SYMBOL_TABLE
"$Revision: 1.101 $"		BOOL	//      $Date: 2008/12/01 14:04:16CET $ $Author: hgc $
"Z_Umlaufzaehler"	C 1	COUNTER	// Temp_Fb242
"Z_Impulszaehler_Motor"	C 9	COUNTER
"Z_min_Takt_Vlies"	C 20	COUNTER	// Minutenzähler für Zwangstakt Vlies
"Z_sec_Takt_Vlies"	C 21	COUNTER	// Sekundenzähler für Zwangstakt Vlies
"Z_MIN_TAKT_SPALTSIEB"	C 22	COUNTER	// Minutenzähler für Intervallbetrieb Spaltsieb
"Z_SEC_TAKT_SPALTSIEB"	C 23	COUNTER	// Sekundenzähler für Intervallbetrieb Spaltsieb
"Z_SPALTSIEB_TAKTE"	C 24	COUNTER	// Zähler für die Spaltsiebtakte
"Z_MSST_COUNT"	C 30	COUNTER
"Z_Schm_FD_War"	C 57	COUNTER
"DB_PLC_MESSAGE"	DB 2	UDT 2	// Schnittstelle für Alarme und Meldungen
"DB_SIEM_GP_DB3"	DB 3	DB 3	// GP SIEMENS
"DB_ALARM_KENNUNG"	DB 4	DB 4	// Siemens Grundprogramm
"DB_SIEM_GP_DB5"	DB 5	DB 5	// GP SIEMENS
"DB_SIEM_GP_DB6"	DB 6	DB 6	// GP SIEMENS
"DB_SIEM_STARTUP"	DB 7	FB 1	// Baseprogram Start-up
"DB_SIEM_SYSTEM4"	DB 8	DB 8	// Baseprogram System
"DB_SIEM_NCK"	DB 10	UDT 10	// Interface NCK
"DB_SIEM_BAG"	DB 11	UDT 11	// Interface BAG
"DB_SINRPC"	DB 12	DB 12	// Interface RPC-PLC
"DB_SIEM_INSTANZ_DB_FB6"	DB 15	FB 6	// GP SIEMENS: Instanz-DB zu FB6
"DB_SIEM_PI"	DB 16	DB 16	// Interface PI-Services
"DB_SIEM_VERSION_CODE"	DB 17	DB 17	// GP SIEMENS: Versionskennung
"DB_SPL"	DB 18	DB 18	// SPL Daten
"DB_SIEM_MMC"	DB 19	UDT 19	// Schnittstelle MMC-Signale
"DB_PLC_MD_DB20"	DB 20	UDT 20	// Maschinenparameter
"DB_SIEM_KANAL_1"	DB 21	UDT 21	// Interface Chanel 1
"DB_SIEM_KANAL_2"	DB 22	UDT 21	// Interface Chanel 2
"DB_ACHSE1_X"	DB 31	UDT 31	// Interface Axis 1 X
"DB_ACHSE2_Y"	DB 32	UDT 31	// Interface Axis 2 Y
"DB_ACHSE3_Z"	DB 33	UDT 31	// Interface Axis 3 Z
"DB_ACHSE4"	DB 34	UDT 31	// Interface Axis 4
"DB_ACHSE5"	DB 35	UDT 31	// Interface Axis 5
"DB_ACHSE6_SPINDEL"	DB 36	UDT 31	// Interface Axis 6 Spindel
"DB_ACHSE7"	DB 37	UDT 31	// Interface Axis 7
"DB_ACHSE8"	DB 38	UDT 31	// Interface Axis 8
"DB_ACHSE9"	DB 39	UDT 31	// Interface Axis 9
"DB_ACHSE10"	DB 40	UDT 31	// Interface Axis 10
"DB_ACHSE11"	DB 41	UDT 31	// Interface Axis 11
"DB_ACHSE12"	DB 42	UDT 31	// Interface Axis 12
"DB_ACHSE13"	DB 43	UDT 31	// Interface Axis 13
"DB_ACHSE14"	DB 44	UDT 31	// Interface Axis 14
"DB_ACHSE15"	DB 45	UDT 31	// Interface Axis 15
"DB_ACHSE16"	DB 46	UDT 31	// Interface Axis 16
"DB_ACHSE17"	DB 47	UDT 31	// Achs Nahtstelle (Achse 17) Simulierte Z-Achse für Komet (U-Achse)
"DB_ACHSE18"	DB 48	UDT 31	// Interface Axis 18
"DB_ACHSE19"	DB 49	UDT 31	// Interface Axis 19
"DB_HR"	DB 50	DB 50	// HR Datenbaustein
"DB_HMI_OEM"	DB 57	DB 57	// OEM Datenbaustein
"DB_HMI"	DB 59	UDT 59	// HMI PRO Datenbaustein
"DB_DEC_HMI"	DB 62	DB 62	// DEC HMI Datenbaustein
"DB_FAMILIEN_MODUL"	DB 65	UDT 65	// Datenbaustein Familienmodul
"DB_TIMER"	DB 66	DB 66	// DB für Timerbaustein
"DB_NC_PLC"	DB 70	UDT 70	// DB für DUAL-Port-RAM: Datentausch NC<==>PLC
"TMLoadIF"	DB 71	UDT 71	// Interface loading-/unloadingstation for Toolmanagment
"TMSpindleIF"	DB 72	UDT 72	// Schnittstelle: Werkzeugverw.: Wechsel in Spindel
"Revolver"	DB 73	UDT 73	// Interface Revolver for Toolmanagment
"DB_OVR_WANDLER"	DB 75	DB 75	// Overridewandler
"DB_DP_DIAG_SINUMERIK"	DB 78	DB 78	// DB DP-Diagnose Sinumerik mit Wizard
"DI_FB_DETAIL_DP_DIAG"	DB 79	FB 96	// Instanz-DB zu FB96
"DB_CMM_PLC"	DB 82	DB 82	// SM PLC-Interface
"DI_FB_PLC_Absturz_GP"	DB 90	FB 29	// Instanz-DB für Diagnose PLC-Absturz im Grundprogramm
"DB_PLC_ABSTURZ_GP_RING"	DB 91	DB 91	// PLC Absturz Grundprogramm
"DB_SIEM_DB_DIAG_DETAIL"	DB 96	FB 96	// Instanz-DB zu FB96 (Transline 200 Anzeige)
"DB_HMI_PRO_RANG_DIAG"	DB 97	DB 97	// Rangierung Diagnosedaten integrierte CP auf HMI-PRO
"DB_DM_PLC_VERSION"	DB 99	DB 99	// Plc Version
"DB_REMANENT"	DB 100	UDT 100	// Remanente Daten
"DB_OEM"	DB 101	DB 101	// OEM-Daten 1
"DB_FEHLERMELDUNG"	DB 102	DB 102	// Fehler- Betriebsmeldungen Maschine
"DB_ANWENDER_SOFTKEY"	DB 103	DB 103	// Anwender Softkeys für Wizard
"DB_EINRICHTFUNKTION"	DB 105	DB 105	// Softkeys für Wizard
"DB_VIB_SCHNITTSTELLE"	DB 106	DB 106	// Schnittstelle Vibrationssensor
"DB_DM_M_FUNKTION"	DB 107	DB 107	// M-Funktionen
"DB_OEMDB2"	DB 108	DB 108	// OEM-Daten 2
"DB_H_FUNKTION"	DB 109	DB 109	// H-Funktionen
"DB_TOOL_DATA"	DB 110	DB 110	// Schneidendaten aktuelles Werkzeug
"DI_GREIFER_DAT_LESEN"	DB 111	FB 2	// Instanz-DB Spindeldaten
"DB_INST_TOOL_DAT"	DB 112	FB 2	// Instanz-DB Schneidendaten
"DI_FB2_VIB_SPI_DATA"	DB 113	FB 2	// Instanz-DB Vibrationssensor
"DI_H_DEKODER"	DB 117	FB 511	// Instanz-DB H-Dekoder
"Schnittstelle_HAWE"	DB 118	DB 118	// Schnittstelle HAWE
"DI_M_DEKODER"	DB 119	FB 510	// Instanz M-Dekoder
"DB_NC_VAR"	DB 120	DB 120	// NC-Variablen DB
"DB_GREIFER_DATEN"	DB 121	DB 121	// Greiferdaten
"DI_OEM_DATEN_GREIFERWZ"	DB 122	FB 2
"DI_GREIFER_DAT_LESEN2"	DB 123	FB 2	// Instanz-DB Greiferdaten lesen 2
"DB_PrgAnwahl"	DB 124	DB 124	// Progr. Pruefen bei Autm. PW
"DB_PAL_PRG_NR"	DB 125	DB 125	// Programm-Nummer
"DI_GET_RESTWEG"	DB 127	FB 2	// Instanz-DB Restweg
"DI_SPI_DATA2"	DB 128	FB 2	// Instanz-DB Spindeldaten 2
"DI_Wz_sperren"	DB 131	FB 131	// Instanz-DB für Werkzeug sperren
"DB_TOOL_DATA _SPEICHER"	DB 137	DB 137	// Werkzeugdatenspeicher
"DB_SPDL_Komp"	DB 138	DB 138	// Datenbaustein Glaettung Kompensation
"DB_Restweg"	DB 140	DB 140	// Restweg
"DB_INST_FB4_ll"	DB 145	FB 4	// Instanz-DB zu FB4
"PRGAnwahl"	DB 146	DB 146	// String für Makro anwahl zum PW
"DB_STERN_DREIECK"	DB 150	DB 150	// Spindel Stern-Dreieck
"DB_WORKPIECE_COUNTER"	DB 152	FB 152	// instance DB for work piece counter
"DB_CYCLE_TIME"	DB 153	FB 153	// instance DB for cycle time measurement
"DB_GETRIEBEUEBERWACH"	DB 156	DB 156
"DI_GETRIEBEUEBERWACHUNG"	DB 157	FB 2
"DB_HMI_PRO_ADDITIONAL"	DB 159	UDT 159	// HMI-PRO: Erweiterung Zähler
"DB_ACHS13_WZM2"	DB 160	DB 160	// Achse 13 WZM2 Zusatzdaten
"DB_ACHS7_WZM"	DB 161	DB 161	// Achse 7 WZM Zusatzdaten
"DB_ACHS13_WZM_Gantry"	DB 162	DB 162	// Achse 13 WZM Gantry-Achse Kette 180 Zusatzdaten
"DB_Achs8"	DB 163	DB 163	// Achse 8 Zusatzdaten
"DB_Achs5"	DB 165	DB 165	// Achse 5 Zusatzdaten
"DB_ACHSE_WZW_QUER"	DB 166	DB 166	// Achse Querhub Werkzeugwechsler
"DB_ACHSE_WZW_LAENGS"	DB 167	DB 167	// Achse längs Werkzeugwechsler
"DB_ACHSE_RPL"	DB 168	DB 168	// Achse 15 Zusatzdaten: drehbare Rüstplatz-Achse
"DI_HANDSHAKE_WZREGAL"	DB 170	FB 170	// Instanz-DB Handshake Werkzeugregal
"DB_IN"	DB 171	DB 171	// Kommunikation - Eingänge
"DB_OUT"	DB 172	DB 172	// Kommunikation - Ausgänge
"Sonder_Datenaustausch"	DB 173	DB 173	// Sonderdatenaustausch
"DI_WZV_ABL_REGAL"	DB 174	FB 174	// Instanz-DB Regal Ablauf
"DB_VWWZ"	DB 175	UDT 175	// Daten für vert. WzWechsler Grundstlg.fahren
"DB_WWZ"	DB 176	UDT 176	// Daten für WzWechsler Grundstlg.fahren
"DB_WW"	DB 177	DB 177	// Werkzeugwechsler
"DI_WZ_BRUCH"	DB 178	FB 178	// Instanz-DB FB_WZ_BRUCH
"DB_WZV"	DB 179	DB 179	// Werkzeugverwaltung
"DB_PW_DATA"	DB 182	DB 182	// Palettenwechsler Daten
"DI_WK_ABLAUF"	DB 184	FB 184	// Instanz-DB Winkelfraeskopf Ablauf
"DI_PW_ABLAUF"	DB 187	FB 187	// Instanz-DB Palettenwechsler Ablauf
"DB_TM_VAR"	DB 190	DB 190	// NC-Variablenliste für Leerplatzsuche
"DI_TM_LEERPLATZ"	DB 191	FB 191	// Instanz-DB FB191 Leerplatz suchen
"DI_TM_MAGDAT"	DB 192	FB 192	// Instanz-DB Magazindaten
"DI_TM_T_BEFEHL"	DB 193	FB 193	// Instanz-DB FB193 T-Befehl auswerten
"DI_TM_QUITT_FC8"	DB 195	FB 195	// Instanz-DB FB195 Quittieren mit FC8
"DI_TM_WZTYP_RD"	DB 196	FB 196	// Instanz-DB Werkzeugtyp RD
"DI_TM_WZBRUCH_R"	DB 197	FB 197	// Instanz-DB Werkzeugbruch lesen
"DI_FB_TM_WZDAT"	DB 198	FB 198	// Instanz-DB für Werkzeugdaten lesen
"DI_TM_QTEST"	DB 199	FB 199	// Instanz-DB Aufzeichnen der Quittierungen
"DB_ASUP_MACHINE"	DB 201	UDT 201	// ASUP Maschine
"DI_GE_SPEZIFIKATION"	DB 202	FB 202	// Instanz-DB für FB GE Spezifikation
"DI_PW_ZUR_GRD"	DB 204	FB 204	// Instanz-DB für FB_PW_ZUR_GRD
"DB_JOB_SORTIERT"	DB 206	DB 206
"DI_KOMET_U_ACHSE"	DB 207	FB 207	// Instanz-DB für FB_KOMET_U_Achse
"DB_RPL_Positionen"	DB 208	DB 208	// Positionen Rüstplatzachse
"DB_CTS"	DB 209	DB 209	// Schnittstelle Werkzeugverwaltung zu CTS
"DB_PI_Service"	DB 210	FB 4	// Instanz-DB PI-Services 1: select ASUP
"DB_JOB"	DB 211	DB 211	//  Daten der Jobliste
"DB_STRINGPW"	DB 212	DB 212	// Palettenwechsler String für Makroanwahl
"DB_SPEICHERTRANSPORT"	DB 213	DB 213	// Speicher Transport
"DB_PAL_NR"	DB 214	DB 214	// Paletten-Nummer
"DB_LSSchnittstelle"	DB 215	DB 215	// Schnittstelle zu LS6
"DB_LS_POS"	DB 216	DB 216	// Linearspeicher Positionen
"DB_Achs9_DrehSt"	DB 217	DB 217	// Achse 9 Palettenspeicher Drehstation Zusatzdaten
"DB_Achs10_Transport"	DB 218	DB 218	// Achse 10 Palettenspeicher Transport Zusatzdaten
"DB_Achs16_Hub_PS"	DB 219	DB 219	// Achse 10 Palettenspeicher Hub Zusatzdaten
"DI_FB_SPH"	DB 220	FB 230	// Instanz-DB Spannhydraulik Funktionen
"DI_FB_Norm_AnalogA"	DB 221	FB 254	// Instanz-DB Normierung eines analogen Ausgang
"DB_Achs11_VMAG_Greifer"	DB 222	DB 222	// Achse 14 Vertikalmagazin Greifer Zusatzdaten
"DI_TM_Get_TNR"	DB 223	FB 200	// Instanz-DB Werkzeugnummer
"DB_TDS"	DB 224	DB 224	// TDS-Balluf
"DI_FB_WZV_Komm"	DB 225	FB 175	// Instanz-DB FB_WZV_Komm (FB175)
"DB_WZV_NCVAR"	DB 226	DB 226	// WZV-NC-Var-Selector
"DB_WZV_DV"	DB 227	DB 227	// WZV-Datenverteiler
"DB_KONFIG_DMTDC"	DB 228	DB 228	// Konvertierungstabelle
"DB_VGL_DMTDC"	DB 229	DB 229	// TDC
"DI_TDC_DM"	DB 230	FB 81	// Instanz-DB
"DI_SIEM_GET_AX7_AX8"	DB 231	FB 2	// Instanz-DB Lesen  Istpositionen Achse 7 und Achse 8
"DI_SIEM_GET_AX16"	DB 232	FB 2	// Instanz-DB Lesen  Istpositionen Achse 16
"DI_SIEM_GET_AX10"	DB 233	FB 2	// Instanz-DB für FB_SIEM_GET: Lesen Istpositionen Achse 10
"DB_UT_UHRZEIT"	DB 234	DB 234	// Uhrzeit
"DI_SIEM_GET_AX9"	DB 235	FB 2	// Instanz-DB für FB_SIEM_GET Maschinendaten Achse 9 lesen
"DI_SIEM_GET_AX15"	DB 236	FB 2	// Instanz-DB für FB_SIEM_GET Achse 15 (Rüstplatz) lesen
"DI_FB_SPH_FD"	DB 237	FB 237	// Instanz-DB für FB_SPH_FD
"DI_SIEM_GET_AX16_SW_CAM"	DB 238	FB 2	// Instanz-DB Lesen  Istpositionen Achse 16 Softwarenocken
"DI_FB_SPH_OPW"	DB 239	FB 239	// Instanz-DB für FB SpannHydraulik OHNE PW
"DB_MSG_AEND"	DB 240	UDT 240	// Erkennung neue Fehler im Db102
"DB_TEMP_KOMP"	DB 241	DB 241	// TEMPERATURKOMPENSATION
"DI_FB_IF_FASTEMS"	DB 243	FB 243	// Instanz-DB
"DB_BALLUFF_BISF"	DB 244	DB 244
"DI_RS232"	DB 245	FB 245
"DI_SIEM_GET_AX14"	DB 246	FB 2	// Instanz-DB lesen Istposition Achse 14
"DI_SIEM_GET_AX18"	DB 247	FB 2	// Instanz-DB lesen Istposition Achse 18
"DI_SIEM_GET_AX19"	DB 248	FB 2	// Instanz-DB lesen Istposition Achse 19
"DB_WORKPIECE_IDENT"	DB 249	DB 249
"DB_COMM_WZREGAL"	DB 250	DB 250	// Werkzeugregal
"DB_SCHNITTST_OMRON"	DB 251	DB 251	// Schnittstelle OMRON
"DB_ALG"	DB 254	UDT 254	// allgemeine Signale
"DB_PLC_OFF_B_AX_KL"	DB 257	DB 257	// PLC Offset für die B-Achs Klemmung
"DB_KMTL_KNOLL"	DB 258	DB 258	// Kühlmittel KNOLL
"DB_Temp_Comp"	DB 260	DB 260	// DMTemperaturkompensation
"DI_TEMP_SPINDEL"	DB 261	FB 211	// Instanz-DB Temperaturkompensation Spindel
"DI_TEMP_TISCH"	DB 262	FB 212	// Instanz-DB Temperaturkompensation Tisch
"DI_TEMP_TAB_SPINDEL"	DB 263	FB 213	// Instanz-DB Temperaturkompensation Tabellen Spindel
"DI_TEMP_TAB_TISCH"	DB 264	FB 214	// Instanz-DB Temperaturkompensation Tabellen Tisch
"DI_DIAG_ANA_IN_PT100"	DB 266	FB 216	// Instanz-DB PT100 Temperaturfühler
"DB_FM_GERI"	DB 267	DB 267	// Fehler- Betriebsmeldungen Maschine
"DB_WZVS"	DB 268	DB 268	// Werkzeugverschleisskontrolle
"DI_TEMP_KTY_TRANSMIT"	DB 269	FB 215	// Instanz-DB KTY Temperaturfühler
"DB_UPPERSCREEN_COMM"	DB 270	DB 270	// Upperscreen Interface Communication
"DB_PV_res2"	DB 271	DB 271	// Palettenverwaltung: res 2
"DB_PV_res3"	DB 272	DB 272	// Palettenverwaltung: res 3
"DB_PV_res4"	DB 273	DB 273	// Palettenverwaltung: res 4
"DB_PV_res5"	DB 274	DB 274	// Palettenverwaltung: res 5
"DB_PV_res6"	DB 275	DB 275	// Palettenverwaltung: res 6
"DB_TEST_TEMPKOMP_VERS"	DB 279	DB 279	// DB Test Temperaturkompensation für Versuch
"DI_FB_WIKO_ABLAUF"	DB 280	FB 185	// Instanz-DB Nahtstelle für Wiegenfräskopf
"DB_ML_SPI"	DB 282	FB 282	// Daten Minimalmengenschmierung Fa.Vogel
"DI_SPI_GLAETT"	DB 285	FB 285
"DI_SMARTKEY"	DB 286	FB 286	// Instanz-DB Smartkey - Auswertung
"DI_SMARTKEY_COM"	DB 287	FB 287	// Instanz-DB Smartkey - Kommunikation zur Identnummer-Übertragung
"DI_SMARTKEY_TEST"	DB 288	FB 288	// Instanz-DB Smartkey - Test zur Identnummer-Übertragung
"DI_SERVICE_AGENT"	DB 289	FB 219	// Instanz-DB Service Agent
"DB_BHG_MPI"	DB 290	DB 290	// Bedienhandgerät MPI
"DI_FB2_AXwerte"	DB 291	FB 2	// Instanz-DB für BGH Achsenwerte lesen
"DI_FB_SIEM_PI_Fastems"	DB 292	FB 4
"DI_FB_SIEM_PUT_Fastems"	DB 293	FB 3
"DI_FB_SIEM_GETGUD_Fastem"	DB 294	FB 5
"DI_FMS_TOOL_HANDLING"	DB 295	FB 291
"DB_OMRON_KOMMANDO"	DB 298	DB 298	// OMRON Kommando
"DB_ICON"	DB 300	DB 300	// Visualisierung ICON`s
"DB_TEST_WZB"	DB 310	DB 310	// Test Werkzeugbruchkontrolle
"DI_FB3_PS_WRITE_GUD"	DB 312	FB 3	// Schreibe GUD für erweiterte Palettendaten
"DI_FB5_PS_GET_GUD"	DB 313	FB 5	// Hole GUD-Token zum Schreiben der erweiterten Palettendaten
"DB_TEILE_NR"	DB 314	DB 314	// Teilenummer
"DB_PS_ADVANCED_DATA"	DB 315	DB 315	// Erweiterte Palettendaten
"DB_PRG_LISTE"	DB 317	DB 317	// Programmliste
"DB_PV_SpH"	DB 318	DB 318	// Spannhydraulik Daten in der Palettenverwaltung
"DI_VENTIL_2E2A_WZ_RIEGEL"	DB 323	FB 250
"DI_VENTIL_2E2A_Kegrng_VM"	DB 329	FB 250
"DI_VENTIL_2E2A_WZK_GRD"	DB 330	FB 250	// Instanz-DB FB250 Transporteinheit WZK-GRD VM
"DI_VENTIL_2E2A_UBG_MAG"	DB 331	FB 250	// Instanz-DB FB250 Transporteinheit ÜBG-MAG VM
"DI_VENTIL_2E2A_WZ_MAG"	DB 332	FB 250	// Instanz-DB FB250  Werkzeug an Magazinposition VM
"DI_VENTIL_2E2A_WZ_RPL"	DB 333	FB 250	// Instanz-DB FB250  Werkzeug am Rüstplatz VM
"DI_VENTIL_2E2A_WWKlappe"	DB 334	FB 250	// Instanz-DB FB250 Werkzeugwechslerklappe VM
"DI_VENTIL_2E2A_WZ_MAG_RI"	DB 336	FB 250
"DB_INST_FB137"	DB 337	FB 537	// Instanz-DB FB137 GMN-Spindelschmierung
"DI_VENTIL_2E2A_HASYST"	DB 338	FB 250
"DI_VENTIL_2E2A_WIKO_CLA"	DB 339	FB 250
"DI_TEMP_TRANSMITTER"	DB 341	FB 215	// Instanz-DB TK Temperatur-Transmitter
"DI_FB2_RD_MD"	DB 351	FB 2	// Instanz-DB FB2 Maschinendaten lesen
"DI_FB2_RD_NC"	DB 352	FB 2	// Instanz-DB FB2 NC-Daten lesen
"DI_SIEM_PUT_WRITE_GUD"	DB 354	FB 3	// Instanz-DB FB3 Temperatukompensation GUD`s schreiben
"DI_FB3_EXTERNE_NV"	DB 361	FB 3	// Instanz-DB FB3 externe Nullpunktverschiebung schreiben
"DB_INST_FB3_db368"	DB 368	FB 4	// Instanz-DB FB4  ASUP Maschine initialisieren
"DB_INST_FB4_DB374"	DB 374	FB 4	// Instanz-DB FB4  PI-Dienst Ruecksetzen des Kennwortes
"DI_FB5_TEMP_KOMP"	DB 380	FB 5	// Instanz-DB FB5 Temperaturkompenstaion
"DI_TDC_WZ_Sperren"	DB 389	FB 82	// Instanz-DB TDC Werkzeug sperren
"DB_SAFE_GR2_BT1_INST"	DB 390	FB 11	// Instanz-DB FB11Safety Integrated Bremsentest 1 Gruppe 2
"DB_SAFE_BTGR1_INST"	DB 391	FB 11	// Instanz-DB FB11Safety Integrated Bremsentest Gruppe 1
"DB_SAFE_BTGR2_INST"	DB 392	FB 11	// Instanz-DB FB11Safety Integrated Bremsentest Gruppe 2
"DB_SAFE_ZD_INST"	DB 396	FB 85	// Safety Integrated Instanz-DB Zeiten Zwangsdynamisierungen
"DB_SAFE_ZD"	DB 397	DB 397	// Safety Integrated Ablauf Zwangsdynamisierung und Bremsentest
"DB_SAFE_ALLG1"	DB 398	DB 398	// Safety Integrated Alggemein 1
"DB_SLAVE_DIAGNOSE"	DB 399	DB 399	// DP-Slave Diagnose
"DI_SIEM_GET_PrgKontrolle"	DB 400	FB 2	// Instanz-DB für FB_SIEM_GET zum Lesen der aktuellen Programm-Nr
"DB_SPI_ANALOG"	DB 410	DB 410	// Daten analoger Werkzeugspanner
"DB_HASYST_EROWA"	DB 411	DB 411
"DB_HANDLINGSYSTEM_3R"	DB 420	DB 420
"DI_FB_SPH_DIAGNOSE"	DB 434	FB 234	// Instanz-DB für FB_SPH_DIAGNOSE
"DB_IF_ROB_DMC"	DB 450	DB 450	// Schnittstelle Roboter an DMC
"DB_IF_DMC_ROB"	DB 451	DB 451	// Schnittstelle DMC an Roboter
"DB_TESTSTAND"	DB 499	DB 499
"DB_MCP_IO_ANPASSUNG"	DB 500	DB 500	// Anpassung IOs an SIEMENS Maschinensteuertafel
"DI_MAPAL_U_ACHSE"	DB 508	FB 208	// Instanz-DB für FB_MAPAL_U_Achse
"DI_FM_NC"	DB 512	FB 512
"DI_ASUP_CHAN_2"	DB 513	FB 513
"DB_HMI_PRO_OVERVIEW"	DB 561	DB 561	// HMI-PRO: Bildelemente/Textfelder Anlagenübersicht
"DB_HMI_PRO_ANWENDER"	DB 565	DB 565	// HMI-PRO: Anwenderdaten
"DB592_DMTDC_RESERVE"	DB 592	DB 592
"DB593_DMTDC_RESERVE"	DB 593	DB 593
"DB594_DMTDC_RESERVE"	DB 594	DB 594
"DB595_DMTDC_RESERVE"	DB 595	DB 595
"DB_CONFIG"	DB 700	DB 700	// Maschinen Konfigurations-Daten
"DB_ROB_IF"	DB 701	DB 701	// Schnittstelle Roboter-Beladung
"RUN_UP"	FB 1	FB 1	// Startup Baseprogram
"FB_SIEM_GET"	FB 2	FB 2	// GP-PLC 840D: Read NC Variable
"FB_SIEM_PUT"	FB 3	FB 3	// GP-PLC 840D: Write NC Variable
"FB_SIEM_PI"	FB 4	FB 4	// GP-PLC 840D: PI-Services 1: select ASUP
"FB_SIEM_GETGUD"	FB 5	FB 5	// GP-PLC 840D: read GUD-Variable
"FB_SIEM_GEN_PI_SERVICES"	FB 6	FB 6	// GP-PLC 840D: Allgemeine Kommunikation für PI-Dienste
"PI_SERV2"	FB 7	FB 7	// PI-Services 2
"M2N"	FB 9	FB 9	// Several OPs/NCUs
"SI_Relais"	FB 10	FB 10	// Safety Integrated: Relais
"SI_BrakeTest"	FB 11	FB 11	// Safety Integrated: Brake Test
"FB16_PI"	FB 16	FB 16	// GP-PLC 840D:
"FB_SIEM_GP_FB17"	FB 17	FB 17	// GP-PLC 840D:
"FB_SIEM_GP_FB18"	FB 18	FB 18	// GP-PLC 840D:
"FB_SIEM_GP_FB19"	FB 19	FB 19	// GP-PLC 840D:
"HiGraphErrEmitterFB"	FB 20	FB 20	// GP-PLC 840D: HiGraph error diagnostic
"FB_PLC_Absturz_GP"	FB 29	FB 29	// GP-PLC 840D: Diagnose PLC-Absturz im Grundprogramm
"FB30_TL2000"	FB 30	FB 30	// Transline 2000 Bereich
"FB31_TL2000"	FB 31	FB 31	// Transline 2000 Bereich
"FB32_TL2000"	FB 32	FB 32	// Transline 2000 Bereich
"FB33_TL2000"	FB 33	FB 33	// Transline 2000 Bereich
"FB34_TL2000"	FB 34	FB 34	// Transline 2000 Bereich
"FB35_TL2000"	FB 35	FB 35	// Transline 2000 Bereich
"FB36_TL2000"	FB 36	FB 36	// Transline 2000 Bereich
"FB37_TL2000"	FB 37	FB 37	// Transline 2000 Bereich
"FB38_TL2000"	FB 38	FB 38	// Transline 2000 Bereich
"FB39_TL2000"	FB 39	FB 39	// Transline 2000 Bereich
"FB40_TL2000"	FB 40	FB 40	// Transline 2000 Bereich
"FB41_TL2000"	FB 41	FB 41	// Transline 2000 Bereich
"FB42_TL2000"	FB 42	FB 42	// Transline 2000 Bereich
"FB43_TL2000"	FB 43	FB 43	// Transline 2000 Bereich
"FB44_TL2000"	FB 44	FB 44	// Transline 2000 Bereich
"FB45_TL2000"	FB 45	FB 45	// Transline 2000 Bereich
"FB46_TL2000"	FB 46	FB 46	// Transline 2000 Bereich
"FB47_TL2000"	FB 47	FB 47	// Transline 2000 Bereich
"FB48_TL2000"	FB 48	FB 48	// Transline 2000 Bereich
"FB49_TL2000"	FB 49	FB 49	// Transline 2000 Bereich
"FB50_TL2000"	FB 50	FB 50	// Transline 2000 Bereich
"FB51_TL2000"	FB 51	FB 51	// Transline 2000 Bereich
"FB52_TL2000"	FB 52	FB 52	// Transline 2000 Bereich
"FB53_TL2000"	FB 53	FB 53	// Transline 2000 Bereich
"FB54_TL2000"	FB 54	FB 54	// Transline 2000 Bereich
"FB55_TL2000"	FB 55	FB 55	// Transline 2000 Bereich
"FB56_TL2000"	FB 56	FB 56	// Transline 2000 Bereich
"FB57_TL2000"	FB 57	FB 57	// Transline 2000 Bereich
"FB58_TL2000"	FB 58	FB 58	// Transline 2000 Bereich
"FB59_TL2000"	FB 59	FB 59	// Transline 2000 Bereich
"FB60_TL2000"	FB 60	FB 60	// Transline 2000 Bereich
"FB61_TL2000"	FB 61	FB 61	// Transline 2000 Bereich
"FB62_TL2000"	FB 62	FB 62	// Transline 2000 Bereich
"FB63_TL2000"	FB 63	FB 63	// Transline 2000 Bereich
"FB64_TL2000"	FB 64	FB 64	// Transline 2000 Bereich
"FB65_TL2000"	FB 65	FB 65	// Transline 2000 Bereich
"FB66_TL2000"	FB 66	FB 66	// Transline 2000 Bereich
"FB67_TL2000"	FB 67	FB 67	// Transline 2000 Bereich
"FB68_TL2000"	FB 68	FB 68	// Transline 2000 Bereich
"FB69_TL2000"	FB 69	FB 69	// Transline 2000 Bereich
"FB70_TL2000"	FB 70	FB 70	// Transline 2000 Bereich
"FB71_TL2000"	FB 71	FB 71	// Transline 2000 Bereich
"FB72_TL2000"	FB 72	FB 72	// Transline 2000 Bereich
"FB73_TL2000"	FB 73	FB 73	// Transline 2000 Bereich
"FB74_TL2000"	FB 74	FB 74	// Transline 2000 Bereich
"FB75_TL2000"	FB 75	FB 75	// Transline 2000 Bereich
"FB76_TL2000"	FB 76	FB 76	// Transline 2000 Bereich
"FB77_TL2000"	FB 77	FB 77	// Transline 2000 Bereich
"FB78_TL2000"	FB 78	FB 78	// Transline 2000 Bereich
"FB79_TL2000"	FB 79	FB 79	// Transline 2000 Bereich
"FB80_TL2000"	FB 80	FB 80	// Transline 2000 Bereich
"FB_TDC_DM"	FB 81	FB 81	// TDS-System (BALLUFF)
"FB_TDC_WZ_Sperren"	FB 82	FB 82	// TDS-System (BALLUFF): WZ sperren wenn beim Beladen Status gesperrt
"FB81_TL2000"	FB 83	FB 83	// Transline 2000 Bereich
"FB82_TL2000"	FB 84	FB 84	// Transline 2000 Bereich
"FB_SAFE_ZD_MAIN"	FB 85	FB 85	// SAFETY INTEGRATED: Zwangsdynamisisierungen Hauptmodul
"FB_SAFE_RESERVE"	FB 86	FB 86	// SAFETY INTEGRATED: Reserve
"FB87_TL2000"	FB 87	FB 87	// Transline 2000 SPL Bereich
"FB88_TL2000"	FB 88	FB 88	// Transline 2000 SPL Bereich
"FB89_TL2000"	FB 89	FB 89	// Transline 2000 SPL Bereich
"FB90_TL2000"	FB 90	FB 90	// Transline 2000 Bereich
"FB91_TL2000"	FB 91	FB 91	// Transline 2000 Bereich
"FB92_TL2000"	FB 92	FB 92	// Transline 2000 Bereich
"FB93_TL2000"	FB 93	FB 93	// Transline 2000 Bereich
"FB94_TL2000"	FB 94	FB 94	// Transline 2000 Bereich
"FB95_TL2000"	FB 95	FB 95	// Transline 2000 Bereich
"DETAIL_DP_DIAG"	FB 96	FB 96	// DETAIL_DP_DIAG
"FB97_TL2000"	FB 97	FB 97	// Transline 2000 Bereich
"FB98_TL2000"	FB 98	FB 98	// Transline 2000 Bereich
"FB99_TL2000"	FB 99	FB 99	// Transline 2000 Bereich
"FB100_TL2000"	FB 100	FB 100	// Transline 2000 Bereich
"FB101_TL2000"	FB 101	FB 101	// Transline 2000 Bereich
"FB102_TL2000"	FB 102	FB 102	// Transline 2000 Bereich
"FB103_TL2000"	FB 103	FB 103	// Transline 2000 Bereich
"FB104_TL2000"	FB 104	FB 104	// Transline 2000 Bereich
"FB105_TL2000"	FB 105	FB 105	// Transline 2000 Bereich
"FB106_TL2000"	FB 106	FB 106	// Transline 2000 Bereich
"FB107_TL2000"	FB 107	FB 107	// Transline 2000 Bereich
"FB108_TL2000"	FB 108	FB 108	// Transline 2000 Bereich
"FB109_TL2000"	FB 109	FB 109	// Transline 2000 Bereich
"FB110_TL2000"	FB 110	FB 110	// Transline 2000 Bereich
"FB111_TL2000"	FB 111	FB 111	// Transline 2000 Bereich
"FB112_TL2000"	FB 112	FB 112	// Transline 2000 Bereich
"FB113_TL2000"	FB 113	FB 113	// Transline 2000 Bereich
"FB114_TL2000"	FB 114	FB 114	// Transline 2000 Bereich
"FB115_TL2000"	FB 115	FB 115	// Transline 2000 Bereich
"FB116_TL2000"	FB 116	FB 116	// Transline 2000 Bereich
"FB117_TL2000"	FB 117	FB 117	// Transline 2000 Bereich
"FB118_TL2000"	FB 118	FB 118	// Transline 2000 Bereich
"FB119_TL2000"	FB 119	FB 119	// Transline 2000 Bereich
"FB120_TL2000"	FB 120	FB 120	// Transline 2000 Bereich
"FB121_TL2000"	FB 121	FB 121	// Transline 2000 Bereich (Programmanwahl Kanal 1)
"FB122_TL2000"	FB 122	FB 122	// Transline 2000 Bereich (Programmanwahl Kanal 2)
"FB123_TL2000"	FB 123	FB 123	// Transline 2000 Bereich (Programmanwahl Kanal 3)
"FB124_TL2000"	FB 124	FB 124	// Transline 2000 Bereich (Programmanwahl Kanal 4)
"FB125_TL2000"	FB 125	FB 125	// Transline 2000 Bereich
"FB126_TL2000"	FB 126	FB 126	// Transline 2000 Bereich
"FB127_TL2000"	FB 127	FB 127	// Transline 2000 Bereich
"FB128_TL2000"	FB 128	FB 128	// Transline 2000 Bereich
"FB129_TL2000"	FB 129	FB 129	// Transline 2000 Bereich
"FB130_TL2000"	FB 130	FB 130	// Transline 2000 Bereich
"FB_Wz_sperren"	FB 131	FB 131	// DM WZV: Werkzeug sperren
"FB132_TL2000"	FB 132	FB 132	// Transline 2000 Bereich Werkzeugüberwachung
"FB133_TL2000"	FB 133	FB 133	// Transline 2000 Bereich Werkzeugüberwachung
"FB134_TL2000"	FB 134	FB 134	// Transline 2000 Bereich Werkzeugüberwachung
"FB135_TL2000"	FB 135	FB 135	// Transline 2000 Bereich
"FB136_TL2000"	FB 136	FB 136	// Transline 2000 Bereich
"FB137_TL2000"	FB 137	FB 137	// Transline 2000 Bereich
"FB138_TL2000"	FB 138	FB 138	// Transline 2000 Bereich
"FB139_TL2000"	FB 139	FB 139	// Transline 2000 Bereich
"FB140_TL2000"	FB 140	FB 140	// Transline 2000 Bereich
"FB141_TL2000"	FB 141	FB 141	// Transline 2000 Bereich
"FB142_TL2000"	FB 142	FB 142	// Transline 2000 Bereich
"FB143_TL2000"	FB 143	FB 143	// Transline 2000 Bereich
"FB144_TL2000"	FB 144	FB 144	// Transline 2000 Bereich
"FB145_TL2000"	FB 145	FB 145	// Transline 2000 Bereich
"FB146_TL2000"	FB 146	FB 146	// Transline 2000 Bereich
"FB147_TL2000"	FB 147	FB 147	// Transline 2000 Bereich
"FB148_TL2000"	FB 148	FB 148	// Transline 2000 Bereich
"FB149_TL2000"	FB 149	FB 149	// Transline 2000 Bereich
"FB150_TL2000"	FB 150	FB 150	// Transline 2000 Bereich
"FB151_TL2000"	FB 151	FB 151	// Transline 2000 Bereich
"FB_WORKPIECE_COUNTER"	FB 152	FB 152	// Supply for HMI screen: work piece counter
"FB_CYCLE_TIME"	FB 153	FB 153	// Supply for HMI screen: cycle time monitoring
"FB154_TL2000"	FB 154	FB 154	// Transline 2000 Bereich
"FB155_TL2000"	FB 155	FB 155	// Transline 2000 Bereich
"FB156_TL2000"	FB 156	FB 156	// Transline 2000 Bereich
"FB157_TL2000"	FB 157	FB 157	// Transline 2000 Bereich
"FB158_TL2000"	FB 158	FB 158	// Transline 2000 Bereich
"FB159_TL2000"	FB 159	FB 159	// Transline 2000 Bereich
"FB160_TL2000"	FB 160	FB 160	// HMI-PRO: DM Transline 2000 Bereich
"FB161_TL2000"	FB 161	FB 161	// HMI-PRO: DM Transline 2000 Bereich
"FB162_TL2000"	FB 162	FB 162	// HMI-PRO: DM Transline 2000 Bereich
"FB163_TL2000"	FB 163	FB 163	// HMI-PRO: DM Transline 2000 Bereich
"FB164_TL2000"	FB 164	FB 164	// HMI-PRO: DM Transline 2000 Bereich
"FB165_TL2000"	FB 165	FB 165	// HMI-PRO: DM Transline 2000 Bereich
"FB166_TL2000"	FB 166	FB 166	// HMI-PRO: DM Transline 2000 Bereich
"FB167_TL2000"	FB 167	FB 167	// HMI-PRO: DM Transline 2000 Bereich
"FB168_TL2000"	FB 168	FB 168	// HMI-PRO: DM Transline 2000 Bereich
"FB169_TL2000"	FB 169	FB 169	// HMI-PRO: DM Transline 2000 Bereich
"FB_HANDSHAKE_WZREGAL"	FB 170	FB 170	// DM WZV: Handshake Werkzeugregeal
"FB_WZV_ABL_REGAL"	FB 174	FB 174	// DM WZV: Omron Regal Tx Werkzeug vorbereiten
"FB_WZV_Komm"	FB 175	FB 175	// DM WZV: Kommunikation PLC-NC
"FB_WZ_BRUCH"	FB 178	FB 178	// DM WZV: Werkzeugbruch
"FB180_TL2000"	FB 180	FB 180	// Transline 2000 Bereich
"FB181_TL2000"	FB 181	FB 181	// Transline 2000 Bereich (Schrittkette 1)
"FB182_TL2000"	FB 182	FB 182	// Transline 2000 Bereich (Schrittkette 2)
"FB183_TL2000"	FB 183	FB 183	// Transline 2000 Bereich (Schrittkette 3)
"FB_WINKELKOPF_ABLAUF"	FB 184	FB 184	// Ablauf Winkelfraeskopf (eigenes Magazin)
"FB_WIKO_ABLAUF"	FB 185	FB 185	// WIEGENFRÄSSKOPF: Ablauf
"FB186_TL2000"	FB 186	FB 186	// Transline 2000 Bereich (Schrittkette 6)
"FB_PW_ABLAUF"	FB 187	FB 187	// PALETTENWECHSLER: Ablauf
"FB188_TL2000"	FB 188	FB 188	// Transline 2000 Bereich (Schrittkette 8)
"FB189_TL2000"	FB 189	FB 189	// Transline 2000 Bereich (Schrittkette 9)
"FB190_TL2000"	FB 190	FB 190	// Transline 2000 Bereich (Schrittkette 10)
"FB_TM_LEERPLATZ"	FB 191	FB 191	// DM WZV: Leerplatzsuche
"FB_TM_MAGAZINDATEN"	FB 192	FB 192	// DM WZV: Magazindaten lesen
"FB_TM_T_BEFEHL"	FB 193	FB 193	// DM WZV: T-Befehl auswerten
"FB_TM_WZBRUCH_W"	FB 194	FB 194	// DM WZV: Daten für WzBruch schreiben
"FB_TM_QUITT_FC8"	FB 195	FB 195	// DM WZV: Quitieren mit FC 8
"FB_TM_WZTYP_RD"	FB 196	FB 196	// DM WZV: Werkzeugtyp lesen
"FB_TM_WZBRUCH_R"	FB 197	FB 197	// DM WZV: Kennung Wz-Bruch lesen
"FB_TM_WZDAT"	FB 198	FB 198	// DM WZV: Werkzeugdaten lesen
"FB_TM_QTEST"	FB 199	FB 199	// DM WZV: Aufzeichnen der Quittierungen
"FB_TM_Get_TNR"	FB 200	FB 200	// DM WZV: Werkzeugnummer aus WZ-Liste lesen
"FB_GE_SPEZIFIKATION"	FB 202	FB 202	// General Electric Spezifikation P11T12
"FB_PW_ZUR_GRD"	FB 204	FB 204	// PALETTENWECHSLER: Zur Grundstellung fahren
"FB_KOMET_U_ACHSE"	FB 207	FB 207	// Schnittstelle zu U-Achswerkzeug Komet
"FB_MAPAL_U_ACHSE"	FB 208	FB 208	// Schnittstelle zu U-Achswerkzeug Mapal
"FB_TEMP_SPINDEL"	FB 211	FB 211	// TEMPERATURKOMPENSATION: Spindel
"FB_TEMP_TISCH"	FB 212	FB 212	// TEMPERATURKOMPENSATION: Tisch
"FB_TEMP_TAB_SPINDEL"	FB 213	FB 213	// TEMPERATURKOMPENSATION: Tabellen Spindel
"FB_TEMP_TAB_TISCH"	FB 214	FB 214	// TEMPERATURKOMPENSATION: Tabellen Tisch
"FB_TEMP_KTY_TRANSMIT"	FB 215	FB 215	// TEMPERATURFÜHLER-KTY:Temperaturdaten lesen und umrechnen
"FB_TEMP_ANA_IN_PT100"	FB 216	FB 216	// TEMPERATURFÜHLER-PT100: Diagnose Analog_Input
"FB_SERVICE_AGENT"	FB 219	FB 219	// Service Agent
"FB222_TL2000"	FB 222	FB 222	// Transline 2000 Bereich
"FB223_TL2000"	FB 223	FB 223	// Transline 2000 Bereich
"FB_SPH"	FB 230	FB 230	// SPANNHYDRAULIK: Abläufe-Steuerung für SPANNEN / ENTSPANNEN
"FB_SPH_Spannen"	FB 231	FB 231	// SPANNHYDRAULIK: Spannstelle SPANNEN
"FB_SPH_Entspannen"	FB 232	FB 232	// SPANNHYDRAULIK: Spannstelle ENTSPANNEN
"FB_SPH_H_FKT"	FB 233	FB 233	// SPANNHYDRAULIK: Auswertung für H-Funktionen
"FB_SPH_DIAGNOSE"	FB 234	FB 234	// SPANNHYDRAULIK: Diagnose HAWE-Box
"FB_SPH_DIAG_STELLE"	FB 235	FB 235	// SPANNHYDRAULIK: Diagnose Spannstelle
"FB_SPH_res3"	FB 236	FB 236	// SPANNHYDRAULIK: Reserve
"FB_SPH_FD"	FB 237	FB 237	// SPANNHYDRAULIK-FD: für FD-Maschinen
"FB_SPH_FD_H_FKT"	FB 238	FB 238	// SPANNHYDRAULIK-FD: Auswertung für H-Funktionen
"FB_SPH_OPW"	FB 239	FB 239	// SPANNHYDRAULIK: für Maschinen OHNE Palettenwechsler
"FB_IF_FASTEMS"	FB 243	FB 243	// Interface to FASTEMS
"FB_RS232"	FB 245	FB 245
"FB_S_RECV_SI"	FB 246	FB 246	// Standard FB Receive Data
"FB_S_SEND_SI"	FB 247	FB 247	// Standard FB Send Data
"FB_VENTIL_2E2A"	FB 250	FB 250	// DM-MODUL: Bewegung 2E2A mit Endlagenabfrage
"FB_VENTIL_3E2A"	FB 251	FB 251	// DM-MODUL: Bewegung 3E2A mit Endlagenabfrage
"FB_MOTOR_TAKT_3POS"	FB 253	FB 253	// Ansteuerung getakteter Scheibenwischermotor mit 3 Positionen
"FB_Norm_AnalogA"	FB 254	FB 254	// KM: Normierung Analog-Ausgang auf Ober- und Untergrenze
"FB_Norm_Analog_IN"	FB 255	FB 255	// Normierung Analog-Eingang auf Ober- und Untergrenze
"FB261_TL2000"	FB 261	FB 261	// Transline 2000 Bereich
"FB262_TL2000"	FB 262	FB 262	// Transline 2000 Bereich
"FB263_TL2000"	FB 263	FB 263	// Transline 2000 Bereich
"FB264_TL2000"	FB 264	FB 264	// Transline 2000 Bereich
"FB265_TL2000"	FB 265	FB 265	// Transline 2000 Bereich
"FB266_TL2000"	FB 266	FB 266	// Transline 2000 Bereich
"FB267_TL2000"	FB 267	FB 267	// Transline 2000 Bereich
"FB268_TL2000"	FB 268	FB 268	// Transline 2000 Bereich
"FB269_TL2000"	FB 269	FB 269	// Transline 2000 Bereich
"FB270_TL2000"	FB 270	FB 270	// Transline 2000 Bereich
"FB_ML_SPI"	FB 282	FB 282	// FB Minimalmengenschmierung Fa. Vogel
"FB_SPI_GLAETT"	FB 285	FB 285
"FB_SMARTKEY"	FB 286	FB 286	// Smartkey Auswertung
"FB_SMARTKEY_COM"	FB 287	FB 287	// Kommunikation mit PILZ-Smartkey zur Identnummer-Übertragung
"FB_SMARTKEY_TEST"	FB 288	FB 288	// Modul zur Simulation des PILZ-Smartkey zur Identnummer-Übertragung
"FB_FMS_TOOL_HANDLING"	FB 291	FB 291
"FB_CI_M_DEKODER"	FB 510	FB 510	// DM: Dekoder M-Funktionen
"FB_CI_H_Dekoder"	FB 511	FB 511	// DM: Dekoder H-Funktionen
"FB_NC_Fehler_Dekoder"	FB 512	FB 512	// Dekoder für NC Fehler in der PLC
"FB_ASUP_CHAN_2"	FB 513	FB 513
"FB_SP_SCHMIERUNG"	FB 537	FB 537	// Spindelschmierung
"FC_SIEM_GP_FC1"	FC 1	FC 1	// GP-PLC 840D:
"GP_HP"	FC 2	FC 2	// cyclic Baseprogram
"FC_SIEM_GP_PRAL"	FC 3	FC 3	// GP-PLC 840D:Alarmtriggered Baseprogram
"FC_SIEM_GP_FC4"	FC 4	FC 4	// GP-PLC 840D:
"FC_SIEM_GP_FC5"	FC 5	FC 5	// GP-PLC 840D:
"FC_SIEM_TM_CYCL"	FC 6	FC 6	// GP-PLC 840D: Werkzeugverwaltung Zyklischer Baustein
"TM_REV"	FC 7	FC 7	// Transfer for Revolverchange
"FC_SIEM_TM_TRANS"	FC 8	FC 8	// GP-PLC 840D:Transfer for Toolmanagment
"ASUP"	FC 9	FC 9	// asynchronous Subprograms
"FC_SIEM_AL_MSG"	FC 10	FC 10	// GP-PLC 840D:Alarms & Messages
"FC_SIEM_GP_FC11"	FC 11	FC 11	// GP-PLC 840D:
"FC_SIEM_GP_FC12"	FC 12	FC 12	// GP-PLC 840D:
"BHGDisp"	FC 13	FC 13	// Displaycontrol for Handheld Unit
"FC_MSTT_SIGNALS"	FC 14	FC 14	// GP-PLC 840D:
"POS_AX"	FC 15	FC 15	// GP-PLC 840D:Positioning of Linear- and Rotaryaxis
"PART_AX"	FC 16	FC 16	// GP-PLC 840D:Positioning of Partaxis
"FC_SIEM_YDELTA"	FC 17	FC 17	// GP-PLC 840D:Y / Delta Control
"FC_SIEM_SPINCTRL"	FC 18	FC 18	// GP-PLC 840D:Spindlecontrol / Part-, Positioning-axis
"FC_SIEM_MCP_IFM"	FC 19	FC 19	// Siemens Grundprogramm: MCP-Signals to Interface, Variant M
"WRITE_MESSAGE"	FC 20	FC 20	// GP-PLC 840D:Write Message to PLC-Diagnostic Buffer
"FC_SIEM_PLC_NCK"	FC 21	FC 21	// GP-PLC 840D:Quick Datachannel
"TM_DIR"	FC 22	FC 22	// Directioncontrol for Toolmanagment Mag.
"FC_SIEM_MCP_IFM2"	FC 24	FC 24	// MCP-Signals to Interface, Variant small
"FC_SIEM_MCP_IFT"	FC 25	FC 25	// MCP-Signals to Interface, Variant T
"FC_SIEM_HPU_MCP"	FC 26	FC 26	// MCP-Signals of PHG to Interface
"NE_STRNG"	FC 29	FC 29	// Not Equal String
"FC_ACHS_VERWALTUNG"	FC 30	FC 30	// Hauptmodul Achsen
"FC_ACHS_1"	FC 31	FC 31	// Achs Nahtstelle (Achse 1)
"FC_ACHS_2"	FC 32	FC 32	// Achs Nahtstelle (Achse 2)
"FC_ACHS_3"	FC 33	FC 33	// Achs Nahtstelle (Achse 3)
"FC_ACHS_4"	FC 34	FC 34	// Achs Nahtstelle (Achse 4)
"FC_ACHS_5"	FC 35	FC 35	// Achs Nahtstelle (Achse 5)
"FC_ACHS_6"	FC 36	FC 36	// Achs Nahtstelle (Achse 6) Spindel
"FC_ACHS_7"	FC 37	FC 37	// Achs Nahtstelle (Achse 7) Werkzeugmagazin
"FC_ACHS_8"	FC 38	FC 38	// Achs Nahtstelle (Achse 8) Palettenwechsler
"FC_ACHS_9"	FC 39	FC 39	// Achs Nahtstelle (Achse 9) Palettenspeicher Drehachse
"FC_ACHS_10"	FC 40	FC 40	// Achs Nahtstelle (Achse 10) Palettenspeicher Teleskopachse
"FC_ACHS_11"	FC 41	FC 41	// Achs Nahtstelle (Achse 11) NC-Teilapperat
"FC_ACHS_12"	FC 42	FC 42	// Achs Nahtstelle (Achse 12) Komet U-Achse
"FC_ACHS_13"	FC 43	FC 43	// Achs Nahtstelle (Achse 13) Werkzeugmagazin Slaveachse
"FC_ACHS_14"	FC 44	FC 44	// Achs Nahtstelle (Achse 14) Werkzeuggreifer (Vertikalmagazin)
"FC_ACHS_15"	FC 45	FC 45	// Achs Nahtstelle (Achse 15) Rüstplatz
"FC_ACHS_16"	FC 46	FC 46	// Achs Nahtstelle (Achse 16) Palettenspeicher Hubachse
"FC_ACHS_17"	FC 47	FC 47	// Achs Nahtstelle (Achse 17) Simulierte Z-Achse für Komet
"FC_ACHS_18"	FC 48	FC 48	// Achs Nahtstelle (Achse 18) Querhub Werkzeugwechsler
"FC_ACHS_19"	FC 49	FC 49	// Achs Nahtstelle (Achse 19) Längsachse Werkzeugwechsler Doppelkette
"FC50_TL2000"	FC 50	FC 50	// Transline 2000 Bereich
"FC51_TL2000"	FC 51	FC 51	// Transline 2000 Bereich
"FC52_TL2000"	FC 52	FC 52	// Transline 2000 Bereich
"FC53_TL2000"	FC 53	FC 53	// Transline 2000 Bereich
"FC54_TL2000"	FC 54	FC 54	// Transline 2000 Bereich
"FC55_TL2000"	FC 55	FC 55	// Transline 2000 Bereich
"FC56_TL2000"	FC 56	FC 56	// Transline 2000 Bereich
"FC_HMI_PRO_DIRECT_KEYS"	FC 57	FC 57	// Rangierung U-Bedienung
"FC58_TL2000"	FC 58	FC 58	// Transline 2000 Bereich
"FC_HMI_VERSORG"	FC 59	FC 59	// Versorgung der HMI-Bausteine
"FC_MA_MAIN"	FC 60	FC 60	// MA: Hauptmodul Maschine (Grundsignale)
"FC_BETRIEBSARTEN"	FC 61	FC 61	// MA: Betriebsarten
"FC_DEC_HMI"	FC 62	FC 62	// Ausdekodierung Signale HMI
"FC63_TL2000"	FC 63	FC 63	// Transline 2000 Bereich
"FC64_TL2000"	FC 64	FC 64	// Transline 2000 Bereich
"FC65_TL2000"	FC 65	FC 65	// Transline 2000 Bereich
"FC66_TL2000"	FC 66	FC 66	// Transline 2000 Bereich
"FC67_TL2000"	FC 67	FC 67	// Transline 2000 Bereich
"FC68_TL2000"	FC 68	FC 68	// Transline 2000 Bereich
"FC69_TL2000"	FC 69	FC 69	// Transline 2000 Bereich
"FC70_TL2000"	FC 70	FC 70	// Transline 2000 Bereich
"FC_TM_MAG2"	FC 71	FC 71
"FC72_TL2000"	FC 72	FC 72	// Transline 2000 Bereich
"FC73_TL2000"	FC 73	FC 73	// Transline 2000 Bereich
"FC_TM_VERWALTUNG"	FC 74	FC 74	// DM WZV: Werkzeugverwaltung Hauptmodul
"FC_TM_SS_QUIT_PLC"	FC 75	FC 75	// DM WZV: Quittieren
"FC_TM_VERWALTUNG_VM"	FC 76	FC 76	// DM WZV: Werkzeugverwaltung Hauptmodul Vertikal-Magazin
"FC_WZV_TELLER"	FC 78	FC 78	// DM WZV: Werkzeugverwaltung Tellermagazin
"FC_TM_BE_ENTLADEN"	FC 79	FC 79	// DM WZV: Magazin Beladen / Entladen
"FC80_TL2000"	FC 80	FC 80	// Transline 2000 Bereich
"FC_DMTDC_MAGWerte_le"	FC 81	FC 81	// Mag-Ref-Werte zum Beladen mit Tool Dialog System aus Konfig-Makro lesen
"FC_DMTDC_FUNKT"	FC 82	FC 82	// TDS-System (BALLUFF): Funktion
"FC_DMTDC"	FC 83	FC 83	// TDS-System (BALLUFF): Hauptmodul
"FC_DMTDC_SFC21"	FC 84	FC 84	// TDS-System (BALLUFF): Daten ablöschen beim Entladen
"FC_SAFE_MAIN"	FC 85	FC 85	// SAFETY INTEGRATED: Hauptmodul
"FC_SAFE_SPL_PLC"	FC 86	FC 86	// SAFETY INTEGRATED: sichere programmierbare Logik PLC
"FC_SAFE_ALLG"	FC 87	FC 87	// SAFETY INTEGRATED: Auswertung kein Stop an Achsen steht an
"FC88_TL2000"	FC 88	FC 88	// Transline 2000 Bereich
"FC89_TL2000"	FC 89	FC 89	// Transline 2000 Bereich
"FC90_TL2000"	FC 90	FC 90	// Transline 2000 Bereich
"FC91_TL2000"	FC 91	FC 91	// Transline 2000 Bereich
"FC92_TL2000"	FC 92	FC 92	// Transline 2000 Bereich
"FC93_TL2000"	FC 93	FC 93	// Transline 2000 Bereich
"FC94_TL2000"	FC 94	FC 94	// Transline 2000 Bereich
"FC95_TL2000"	FC 95	FC 95	// Transline 2000 Bereich
"FC96_TL2000"	FC 96	FC 96	// Transline 2000 Bereich
"FC_HMI_PRO_RANG_DIAG_DP"	FC 97	FC 97	// DP-Diagnose für interne SST
"FC98_TL2000"	FC 98	FC 98	// Transline 2000 Bereich
"FC99_TL2000"	FC 99	FC 99	// Transline 2000 Bereich
"FC100_TL2000"	FC 100	FC 100	// Transline 2000 Bereich
"FC101_TL2000"	FC 101	FC 101	// Transline 2000 Bereich
"FC102_TL2000"	FC 102	FC 102	// Transline 2000 Bereich
"FC103_TL2000"	FC 103	FC 103	// Transline 2000 Bereich
"FC104_TL2000"	FC 104	FC 104	// Transline 2000 Bereich
"FC_SCALE"	FC 105	FC 105	// Scaling Values
"FC_UNSCALE"	FC 106	FC 106	// Unscaling Values
"FC107_TL2000"	FC 107	FC 107	// Transline 2000 Bereich
"FC108_TL2000"	FC 108	FC 108	// Transline 2000 Bereich
"FC109_TL2000"	FC 109	FC 109	// Transline 2000 Bereich
"BLOCK_FC"	FC 111	FC 111
"FC112_TL2000"	FC 112	FC 112	// Transline 2000 Bereich
"FC113_TL2000"	FC 113	FC 113	// Transline 2000 Bereich
"FC114_TL2000"	FC 114	FC 114	// Transline 2000 Bereich
"FC_BHG"	FC 115	FC 115	// Mini Bedienhandgeraet
"FC_CS_BHG_MPI"	FC 116	FC 116	// Bedienhandgerät MPI für DS-Software
"FC118_TL2000"	FC 118	FC 118	// Transline 2000 Bereich
"FC119_TL2000"	FC 119	FC 119	// Transline 2000 Bereich
"FC120_TL2000"	FC 120	FC 120	// Transline 2000 Bereich
"FC_CHAN1"	FC 121	FC 121	// Kanal 1 Modul
"FC_CHAN2"	FC 122	FC 122	// Kanal 2 Modul
"FC_CHAN3"	FC 123	FC 123	// Kanal 3 Modul
"FC_CHAN4"	FC 124	FC 124	// Kanal 4 Modul
"FC125_TL2000"	FC 125	FC 125	// Transline 2000 Bereich
"FC126_TL2000"	FC 126	FC 126	// Transline 2000 Bereich
"FC127_TL2000"	FC 127	FC 127	// Transline 2000 Bereich
"FC128_TL2000"	FC 128	FC 128	// Transline 2000 Bereich
"FC129_TL2000"	FC 129	FC 129	// Transline 2000 Bereich
"FC130_TL2000"	FC 130	FC 130	// Transline 2000 Bereich
"FC_WZVS_VERWALTUNG"	FC 131	FC 131	// WZVS: Aufrufbaustein für Werkzeugverschleisskontrolle
"FC132_TL2000"	FC 132	FC 132	// Transline 2000 Bereich
"FC133_TL2000"	FC 133	FC 133	// Transline 2000 Bereich
"FC134_TL2000"	FC 134	FC 134	// Transline 2000 Bereich
"FC135_TL2000"	FC 135	FC 135	// Transline 2000 Bereich
"FC_OP_MESSTASTER"	FC 136	FC 136	// OP: Modul fuer Messtaster
"FC_VIBRATIONSSENSOR"	FC 137	FC 137	// VIBRATIONSSENSOR: Auswertung analoges Signal
"FC138_TL2000"	FC 138	FC 138	// Transline 2000 Bereich
"FC139_TL2000"	FC 139	FC 139	// Transline 2000 Bereich
"FC140_TL2000"	FC 140	FC 140	// Transline 2000 Bereich
"FC141_TL2000"	FC 141	FC 141	// Transline 2000 Bereich
"FC142_TL2000"	FC 142	FC 142	// Transline 2000 Bereich
"FC143_TL2000"	FC 143	FC 143	// Transline 2000 Bereich
"FC144_TL2000"	FC 144	FC 144	// Transline 2000 Bereich
"FC145_TL2000"	FC 145	FC 145	// Transline 2000 Bereich
"FC146_TL2000"	FC 146	FC 146	// Transline 2000 Bereich
"FC147_TL2000"	FC 147	FC 147	// Transline 2000 Bereich
"FC148_TL2000"	FC 148	FC 148	// Transline 2000 Bereich
"FC_SAFETY_GATES"	FC 149	FC 149	// Schutztüren
"FC150_TL2000"	FC 150	FC 150	// Transline 2000 Bereich
"FC_HMI_PRO_ADDITION"	FC 151	FC 151	// HMI-PRO: Verwaltung Zusatzbausteine
"FC152_TL2000"	FC 152	FC 152	// Transline 2000 Bereich
"FC153_TL2000"	FC 153	FC 153	// Transline 2000 Bereich
"FC154_TL2000"	FC 154	FC 154	// Transline 2000 Bereich
"FC155_TL2000"	FC 155	FC 155	// Transline 2000 Bereich
"FC156_TL2000"	FC 156	FC 156	// Transline 2000 Bereich
"FC157_TL2000"	FC 157	FC 157	// Transline 2000 Bereich
"FC158_TL2000"	FC 158	FC 158	// Transline 2000 Bereich
"FC159_TL2000"	FC 159	FC 159	// Transline 2000 Bereich
"FC_HMI_PRO_HEADER"	FC 160	FC 160	// HMI-PRO: DM Header
"FC_HMI_PRO_OVERVIEW"	FC 161	FC 161	// HMI-PRO: DM Anlagenübersicht
"FC162_DM_TL2000"	FC 162	FC 162	// HMI-PRO: DM Transline 2000 Bereich
"FC163_DM_TL2000"	FC 163	FC 163	// HMI-PRO: DM Transline 2000 Bereich
"FC164_DM_TL2000"	FC 164	FC 164	// HMI-PRO: DM Transline 2000 Bereich
"FC_HMI_PRO_MANUAL"	FC 165	FC 165	// HMI-PRO: Handfunktionen (Rettung)
"FC_HMI_PRO_RUN_UP"	FC 166	FC 166	// HMI-PRO: Einschaltbedingungen
"FC_HMI_PRO_MODES"	FC 167	FC 167	// HMI-PRO: Taktarten
"FC168_DM_TL2000"	FC 168	FC 168	// HMI-PRO: DM Transline 2000 Bereich
"FC169_DM_TL2000"	FC 169	FC 169	// HMI-PRO: DM Transline 2000 Bereich
"FC170_DM_TL2000"	FC 170	FC 170	// HMI-PRO: DM Transline 2000 Bereich
"FC171_DM_TL2000"	FC 171	FC 171	// HMI-PRO: DM Transline 2000 Bereich
"FC172_DM_TL2000"	FC 172	FC 172	// HMI-PRO: DM Transline 2000 Bereich
"FC173_DM_TL2000"	FC 173	FC 173	// HMI-PRO: DM Transline 2000 Bereich
"FC_HMI_IO_TO_TLINE"	FC 174	FC 174	// HMI-PRO: Zuweisen der IO und Bedingungen an den DB59
"FC_HMI_OEM_TO_TLINE"	FC 175	FC 175	// HMI-PRO: Zuweisung der Daten von OEM DB101 an Transline DB59
"FC_HMI_TLINE_TO_FUNK"	FC 177	FC 177	// HMI-PRO: Bewegungsdaten von Transline DB62 an Einrichtfunktion DB105
"FC_HMI_DEC_TLINE"	FC 178	FC 178	// HMI-PRO: Daten von Transline DB59 an Transline DB62
"FC179_DM_TL2000"	FC 179	FC 179	// HMI-PRO: DM Transline 2000 Bereich
"FC_MANAGE_FUNC_GROUP"	FC 180	FC 180	// Verwaltung der Funktionsgruppen
"FC181_FUNKTIONSGRP_1"	FC 181	FC 181	// FUNKTIONSGRUPPE 1:                                     Reserve
"FC_WZW_VERWALTUNG"	FC 182	FC 182	// WZW: Hauptmodul Werkzeugwechlser Verwaltung
"FC_MAG_VERWALTUNG"	FC 183	FC 183	// MAG: HAuptmodul  Magazinverwaltung
"FC_LASER_VERWALTUNG"	FC 184	FC 184	// LASERVERMESSUNG: Hauptmodul
"FC_WIKO_MAIN"	FC 185	FC 185	// WIEGENFRÄSSKOPF: Hauptmodul
"FC_SK_MAIN"	FC 186	FC 186	// SCHWENKKOPF:Hauptmodul
"FC_PW_VERWALTUNG"	FC 187	FC 187	// PALETTENWECHSLER: Hauptmodul
"FC_PS_MAIN"	FC 188	FC 188	// PALETTENSPEICHER: Hauptmodul
"FC181_FUNKTIONSGRP_9"	FC 189	FC 189	// FUNKTIONSGRUPPE 9:                                     Reserve
"FC_VSM_RPT_CS_Reihe"	FC 190	FC 190	// RUESTPLATZ: Verwaltungs- und SteuerModul für CS-Reihe
"FC_MA_MASCHINE_EIN"	FC 191	FC 191	// MA: Maschine Ein
"FC_MA_HYDRAULIK_EIN"	FC 192	FC 192	// MA: Hydraulik
"FC_MA_PNEUMATIK_EIN"	FC 193	FC 193	// MA: Pneumatik
"FC_MA_SCHMIERUNG"	FC 194	FC 194	// MA: Hauptmodul Schmierung
"FC_MA_SCHMIERZYKLUS"	FC 195	FC 195	// MA: Schmierzyklus
"FC_MA_ALLG_UEBERW"	FC 196	FC 196	// MA: Allgemeine Überwachungen
"FC_MA_SPI_SCHMIER"	FC 197	FC 197	// MA: Spindelschmierung
"FC_MA_PASS_FEI_WAR"	FC 198	FC 198	// MA: Passwort- / Kennwort Reset / Feierabendschaltung
"FC_MA_KUEHLAGGREGAT"	FC 199	FC 199	// MA: Kühlaggregat
"FC_ASUP_MACHINE"	FC 201	FC 201	// ASUP Maschine
"FC_Prg_Anwahl_1"	FC 202	FC 202	// Programmanwahl 1
"STRNG_I"	FC 204	FC 204	// String to Integer
"FC_PRG_Anwahl_Main"	FC 205	FC 205	// Programmanwahl Hauptmodul
"FC_Prg_Anwahl_Check"	FC 206	FC 206	// Programmanwahl Check
"FC_Prg_Job_Suche"	FC 208	FC 208	// Programm Job-Suche
"EQ_STRNG"	FC 209	FC 209	// Equal String
"FC_TEMP_KOMP_MAIN"	FC 210	FC 210	// TEMPERATURKOMPENSATION: Hauptmodul
"FC_TEMP_PT100"	FC 211	FC 211	// TEMPERATURKOMPENSATION: Temperaturerfassung PT100
"FC_TEMP_HILFSFKT"	FC 212	FC 212	// TEMPERATURKOMPENSATION: Hilsfunktion für FB263
"FC_TEMP_WRITE_GUD"	FC 213	FC 213	// TEMPERATURKOMPENSATION: GUD`s schreiben
"FC_TEMP_FUNKTIONEN"	FC 214	FC 214	//  Auswerten von Maschinenparametern INT
"FC_WZVS_MCU"	FC 216	FC 216	// WZVS: Werkzeugverschleiss / Bruch Überwachung mit MCU
"FC_WZVS_ARTIS_MAIN"	FC 217	FC 217	// WZVS: Artis Hauptprogramm
"FC_WZVS_ARTIS"	FC 218	FC 218	// WZVS: Artis Unterprogramm
"FC_SERVICE_AGENT"	FC 219	FC 219	// Service Agent
"FC_220_UT_RESERVE"	FC 220	FC 220	// UT:                                                         Reserve
"FC_UT_CHAR_TO_BYTE"	FC 221	FC 221	// UT: Char to byte
"FC222_TL2000"	FC 222	FC 222	// Transline 2000 Bereich
"FC223_TL2000"	FC 223	FC 223	// Transline 2000 Bereich
"FC_UT_IO_PROFIBUS"	FC 225	FC 225	// UT: E/A-Adressen über PROFIBUS übertragen
"FC_UT_TIMER"	FC 226	FC 226	// UT: Baustein für zusätzliche Timer
"FC_UT_BIT_TO_DEZ"	FC 227	FC 227	// UT: Umwandlung Bit in Dezimal
"FC_UT_SLAVE_UEBERW"	FC 229	FC 229	// UT: Überwachung der Slaves
"FC_UT_STRING_VGL"	FC 230	FC 230	// UT: Vergleichen zweier Strings
"FC_UT_AXIS_READ"	FC 231	FC 231	// UT: Achspositionen lesen
"FC_UT_DYN_UEBW"	FC 232	FC 232	// UT: Dynamische Überwachung
"FC_UT_FKT_Lib"	FC 233	FC 233	// UT: Function Library - DECKEL MAHO Funktions-Bibliothek
"FC_UT_GRAY_TO_BIN"	FC 234	FC 234	// UT: Umwandlung Greycode to Binary
"FC_UT_ANWENDER_SK"	FC 236	FC 236	// UT: Softkey Anwender Funktionen
"FC_237_UT_RESERVE"	FC 237	FC 237
"FC_UT_Bit_auf_Byte"	FC 239	FC 239	// UT: Bit auf Byte
"FC_OP_Main"	FC 240	FC 240	// OP: Verwaltung
"FC_OP_SPAE_SPUE"	FC 243	FC 243	// OP: Modul fuer Spaenefoerderer, Spuelpistole
"FC_OP_M190"	FC 244	FC 244	// OP: M190 Modul
"FC_OP_CODE_M18x"	FC 245	FC 245	// OP: M180-M189 Modul
"FC_OPERATOR_GUIDANCE"	FC 246	FC 246	// Bedienerführung
"FC_SIGNALLEUCHTE"	FC 247	FC 247	// Signalleuchte ROT/GELB/GRÜN/BLAU
"FC_B_KOMP"	FC 248	FC 248	// Kompensation B-Achse
"FC_FAMILIEN_MODUL"	FC 250	FC 250	// Familienmodul
"FC_FAM_M_RESET"	FC 251	FC 251	// Reset unbenützte M-Funktionsmerker
"FC_ZYLINDER"	FC 252	FC 252	// Unterprogramm fuer einen Zylinder
"FC_DISPLAY_ICONS"	FC 253	FC 253	// Anzeige der Icons in der Headerleiste Maschine
"FC_DISPLAY_DMGHEADER"	FC 254	FC 254	// Baustein zur Anzeige der Icons im DMG-Header
"FC261_TL2000"	FC 261	FC 261	// Transline 2000 Bereich
"FC262_TL2000"	FC 262	FC 262	// Transline 2000 Bereich
"FC263_TL2000"	FC 263	FC 263	// Transline 2000 Bereich
"FC264_TL2000"	FC 264	FC 264	// Transline 2000 Bereich
"FC265_TL2000"	FC 265	FC 265	// Transline 2000 Bereich
"FC266_TL2000"	FC 266	FC 266	// Transline 2000 Bereich
"FC267_TL2000"	FC 267	FC 267	// Transline 2000 Bereich
"FC268_TL2000"	FC 268	FC 268	// Transline 2000 Bereich
"FC269_TL2000"	FC 269	FC 269	// Transline 2000 Bereich
"FC270_TL2000"	FC 270	FC 270	// Transline 2000 Bereich
"FC_KUEHLMITTEL"	FC 271	FC 271	// KM: Hauptmodul Kuehlmittel
"FC_IKZ_ANALOG_DRUCK"	FC 272	FC 272	// KM: IKZ-Hochdruckanlage mit variablen Druckstufen
"FC_IKZ_DRUCKSTUFEN"	FC 273	FC 273	// KM: Druckstufen innere Kühlmittelzufuhr
"FC_IKZ_UEBERWACHUNG"	FC 274	FC 274	// KM: Durchfluss-Überwachung für Kühlmittel-Hochdruck (IKZ /  M7)
"FC_KMTL_KSA7"	FC 275	FC 275	// KM: BLECHTECHNIK Spaltsiebanlage gesteuert gereinigt
"FC_KMTL_KSA3"	FC 276	FC 276	// KM: BÜRENER Bandfilterkühlmittelanlage
"FC_KMTL_KSA3.1"	FC 277	FC 277	// KM: BÜRENER Bandfilterkühlmittelanlage mit Zusatzpäneförderer
"FC_KMTL_KNOLL"	FC 278	FC 278	// KM: KNOLL Kuehlmittelanlage VRF250
"FC_KMTL_KSA4"	FC 279	FC 279	// KM: INTERLIT Kuehlmittelanlage mit Kratzförderer
"FC_ZEIT_DIFF"	FC 280	FC 280	// SPINDELSCHMIERUNG: Zeitdifferenz Systemzeit <-> letzter Schmiervorgang
"CONCAT"	FC 281	FC 281	// Concatenate  String
"DI_STRNG"	FC 282	FC 282	// Double Integer to String
"FC_SAFE_ZD1_6AX1"	FC 285	FC 285	// SAFETY INTEGRATED: Zwangsdynamisierung der Abschaltpfade (6Achsen)
"FC_SAFE_ZD2_8AX1"	FC 286	FC 286	// SAFETY INTEGRATED: Zwangsdynamisierung der externen Stopps (8Achsen)
"FC_SAFE_ZD_BER2_PS"	FC 287	FC 287	// SAFETY INTEGRATED: Zwangsdynamisierung Bereich 2 -  Palettenspeicher (PS/PW)
"FC_SAFE_ZD_BER1_MA"	FC 288	FC 288	// SAFETY INTEGRATED: Zwangsdynamisierung Bereich 1 -  Maschine (ARB/ WZW/PW)
"FC_DIAG_SICHERN"	FC 289	FC 289	// SAFETY INTEGRATED:: DP-Slavediagnose sichern
"FC_OVR_PROZENT"	FC 290	FC 290	// Override Prozent
"FC_SINRPC"	FC 292	FC 292	// SINRPC
"FC_RP_VSKORR"	FC 293	FC 293	// GeschwKorr. für RpAchse aus Poti und 4 Bit ADU
"FC_FMS_MC_IF"	FC 294	FC 294
"FC_DP_DIAG_SINUMERIK"	FC 297	FC 297	// DP-Diagnoseanbindung an Sinumerik (Wizard)
"FC300_FKT_GRP_1"	FC 300	FC 300	// Funktionsgruppe 1                                                    Reserve
"FC301_FKT_GRP_1"	FC 301	FC 301	// Funktionsgruppe 1                                                    Reserve
"FC302_FKT_GRP_1"	FC 302	FC 302	// Funktionsgruppe 1                                                    Reserve
"FC303_FKT_GRP_1"	FC 303	FC 303	// Funktionsgruppe 1                                                    Reserve
"FC304_FKT_GRP_1"	FC 304	FC 304	// Funktionsgruppe 1                                                    Reserve
"FC305_FKT_GRP_1"	FC 305	FC 305	// Funktionsgruppe 1                                                    Reserve
"FC306_FKT_GRP_1"	FC 306	FC 306	// Funktionsgruppe 1                                                    Reserve
"FC307_FKT_GRP_1"	FC 307	FC 307	// Funktionsgruppe 1                                                    Reserve
"FC308_FKT_GRP_1"	FC 308	FC 308	// Funktionsgruppe 1                                                    Reserve
"FC309_FKT_GRP_1"	FC 309	FC 309	// Funktionsgruppe 1                                                    Reserve
"FC_WZW_ABLAUF"	FC 310	FC 310	// WZW: Ablaufmodul
"FC_WZW_STATUS"	FC 311	FC 311	// WZW: Statusmodul
"FC_WZW_FEHLER"	FC 312	FC 312	// WZW: Fehlermodul
"FC313_WZW_RESERVE"	FC 313	FC 313	// WZW:                                                                     Reserve
"FC_WZ_SPANNER"	FC 314	FC 314	// WZW: Werkzeugspanner
"FC_KEGELREINIGUNG"	FC 315	FC 315	// WZW: Kegelreinigung 60S
"FC_KEGELREINIGUNG_VM"	FC 316	FC 316
"FC318_WZW_RESERVE"	FC 318	FC 318	// WZW:                                                                     Reserve
"FC_MWZW_Ablauf"	FC 319	FC 319	// WZW: manueller Werkzeugwechsel-Ablauf
"FC320_WZW_RESERVE"	FC 320	FC 320	// WZW:                                                                     Reserve
"FC_WZW_VMAG_STATUS"	FC 321	FC 321	// WZW: Vertikal-Magazin-Wechsler: Status
"FC_WW_TELLER"	FC 322	FC 322	// WZW: Werkzeugwechsler Teller
"FC_WZW_VERT_MAG"	FC 323	FC 323	// WZW: Baustein für Vertikal-Magazin-Wechsler
"FC_WMT_POSITIONIEREN"	FC 324	FC 324	// WZW:  Werkzeugwechsler Teller positionieren
"FC325_WZW_RESERVE"	FC 325	FC 325	// WZW:                                                                     Reserve
"FC_WW_SCHRITT_GEN"	FC 326	FC 326	// WZW: Schrittgenerierung
"FC327_WZW_RESERVE"	FC 327	FC 327	// WZW:                                                                     Reserve
"FC_WW_SPANNER"	FC 328	FC 328	// WZW: Spanner
"FC329_WZW_RESERVE"	FC 329	FC 329	// WZW:                                                                     Reserve
"FC330_WZW_RESERVE"	FC 330	FC 330	// WZW:                                                                     Reserve
"FC_WZW_GREIFER_AUSF"	FC 331	FC 331	// WZW: Greifer aus- einfahren
"FC332_WZW_RESERVE"	FC 332	FC 332	// WZW:                                                                     Reserve
"FC333_WZW_RESERVE"	FC 333	FC 333	// WZW:                                                                     Reserve
"FC334_WZW_RESERVE"	FC 334	FC 334	// WZW:                                                                     Reserve
"FC335_WZW_RESERVE"	FC 335	FC 335	// WZW:                                                                     Reserve
"FC336_WZW_RESERVE"	FC 336	FC 336	// WZW:                                                                     Reserve
"FC_WZB_FSTRT"	FC 337	FC 337	// WZW: Werkzeugbruchüberwachung Frühstart
"FC_WZB_Lesen"	FC 338	FC 338	// WZW: Werkzeugbruchüberwachung lesen
"FC_WZB_TEST"	FC 339	FC 339	// WZW: Werkzeugbruchüberwachung Test
"FC340_MAG_RESERVE"	FC 340	FC 340	// MAG:                                                                     Reserve
"FC341_MAG_RESERVE"	FC 341	FC 341	// MAG:                                                                     Reserve
"FC_GR_MAG"	FC 342	FC 342	// MAG: Ablaufmodul geregeltes Magazin
"FC_GT_MAG_STAT"	FC 343	FC 343	// MAG: Status getaktetes Magazin
"FC_GT_MAG_ABL"	FC 344	FC 344	// MAG: Ablaufmodul getaktetes Magazin
"FC_MAG_HAUPT_ZH"	FC 345	FC 345	// MAG: Hauptmodul / Zweihandbedienung
"FC346_MAG_RESERVE"	FC 346	FC 346	// MAG:                                                                     Reserve
"FC347_MAG_RESERVE"	FC 347	FC 347	// MAG:                                                                     Reserve
"FC348_MAG_RESERVE"	FC 348	FC 348	// MAG:                                                                     Reserve
"FC349_MAG_RESERVE"	FC 349	FC 349	// MAG:                                                                     Reserve
"FC350_LASER_RESERVE"	FC 350	FC 350	// LASER:                                                                  Reserve
"FC351_LASER_RESERVE"	FC 351	FC 351	// LASER:                                                                  Reserve
"FC352_LASER_RESERVE"	FC 352	FC 352	// LASER:                                                                  Reserve
"FC353_LASER_RESERVE"	FC 353	FC 353	// LASER:                                                                  Reserve
"FC354_LASER_RESERVE"	FC 354	FC 354	// LASER:                                                                  Reserve
"FC355_LASER_RESERVE"	FC 355	FC 355	// LASER:                                                                  Reserve
"FC356_LASER_RESERVE"	FC 356	FC 356	// LASER:                                                                  Reserve
"FC357_LASER_RESERVE"	FC 357	FC 357	// LASER:                                                                  Reserve
"FC358_LASER_RESERVE"	FC 358	FC 358	// LASER:                                                                  Reserve
"FC_KALIBRIERRING"	FC 359	FC 359	// OP: Modul fuer Kalibrierring
"FC_WIKO_SS-PS"	FC 360	FC 360	// WIEGENFRÄSSKOPF: Schnittstelle Palettenspeicher
"FC_WiKo_Trans_Abfrage"	FC 361	FC 361	// WIEGENFRÄSSKOPF: Transportabfrage
"FC_WiKo_Abfr_Ueb"	FC 362	FC 362	// WIEGENFRÄSSKOPF: FC_WiKo_Abfr_Ueb
"FC363_WIKO_RESERVE"	FC 363	FC 363	// WIEGENFRÄSSKOPF                                              Reserve
"FC364_WIKO_RESERVE"	FC 364	FC 364	// WIEGENFRÄSSKOPF                                              Reserve
"FC365_WIKO_RESERVE"	FC 365	FC 365	// WIEGENFRÄSSKOPF                                              Reserve
"FC366_WIKO_RESERVE"	FC 366	FC 366	// WIEGENFRÄSSKOPF                                              Reserve
"FC367_WIKO_RESERVE"	FC 367	FC 367	// WIEGENFRÄSSKOPF                                              Reserve
"FC368_WIKO_RESERVE"	FC 368	FC 368	// WIEGENFRÄSSKOPF                                              Reserve
"FC369_WIKO_RESERVE"	FC 369	FC 369	// WIEGENFRÄSSKOPF                                              Reserve
"FC_SK_Ablauf"	FC 370	FC 370	// SCHWENKKOPF:Ablaufmodul
"FC_SK_Status"	FC 371	FC 371	// SCHWENKKOPF:Statusmodul
"FC_SK_FehlerUe"	FC 372	FC 372	// SCHWENKKOPF:Fehlerueberwachung
"FC_SK_X-Fahrbereich"	FC 373	FC 373	// SCHWENKKOPF:Fahrbereiche X-Achse / Stellung B-Kopf
"FC374_SK_RESERVE"	FC 374	FC 374	// SCHWENKKOPF:                                                    Reserve
"FC375_SK_RESERVE"	FC 375	FC 375	// SCHWENKKOPF:                                                    Reserve
"FC376_SK_RESERVE"	FC 376	FC 376	// SCHWENKKOPF:                                                    Reserve
"FC377_SK_RESERVE"	FC 377	FC 377	// SCHWENKKOPF:                                                    Reserve
"FC378_SK_RESERVE"	FC 378	FC 378	// SCHWENKKOPF:                                                    Reserve
"FC379_SK_RESERVE"	FC 379	FC 379	// SCHWENKKOPF:                                                    Reserve
"FC380_PW_RESERVE"	FC 380	FC 380	// PALETTENWECHSLER:                                          Reserve
"FC_PW_AUTOMATIK"	FC 381	FC 381	// PALETTENWECHSLER: Automatikablauf
"FC_PW_FEHLERMODUL"	FC 382	FC 382	// PALETTENWECHSLER: Fehlerüberwachung
"FC_PW_SCHMIERUNG"	FC 383	FC 383	// PALETTENWECHSLER: Schmierung Führungsrohr PW-Hub bei SRT
"FC_RANGIER_PW_DATA1"	FC 384	FC 384	// PALETTENWECHSLER: Datentausch
"FC_PV_PRGlesen_NC"	FC 385	FC 385	// PALETTENWECHSLER: Lesen der Programmnummer von NC
"FC386_PW_RESERVE"	FC 386	FC 386	// PALETTENWECHSLER:                                          Reserve
"FC387_PW_RESERVE"	FC 387	FC 387	// PALETTENWECHSLER:                                          Reserve
"FC388_PW_RESERVE"	FC 388	FC 388	// PALETTENWECHSLER:                                          Reserve
"FC389_PW_RESERVE"	FC 389	FC 389	// PALETTENWECHSLER:                                          Reserve
"FC_PS_PALVERWALTUNG"	FC 390	FC 390	// PALETTENSPEICHER: Palettenverwaltung
"FC_PS_FehlUebw"	FC 391	FC 391	// PALETTENSPEICHER: Fehlerüberwachung
"FC392_PS_RESERVE"	FC 392	FC 392	// PALETTENSPEICHER:                                          Reserve
"FC_PS_RS4_5_SKR"	FC 393	FC 393	// PALETTENSPEICHER: RS4 / RS5 Rettungsfunktion
"FC_PS_RS4_5_ABLAUF"	FC 394	FC 394	// PALETTENSPEICHER: RS4/RS5 Ablauf
"FC_PS_DrehSt_Pos"	FC 395	FC 395	// PALETTENSPEICHER: Drehstation positionieren
"FC_PS_Transp_Pos"	FC 396	FC 396	// PALETTENSPEICHER: Transport positionieren
"FC_PS_Check_Transport"	FC 397	FC 397	// PALETTENSPEICHER: Transport überprüfen
"FC_PS_Pal_Auftr"	FC 398	FC 398	// PALETTENSPEICHER: Palettenauftrag
"FC399_PS_RESERVE"	FC 399	FC 399	// PALETTENSPEICHER:                                           Reserve
"FC_PS_SpeicherzuMa"	FC 400	FC 400	// PALETTENSPEICHER: Transportauftrag Speicher zur Maschine
"FC_PS_MazuSpeicher"	FC 401	FC 401	// PALETTENSPEICHER: Transportauftrag Maschine zum Speicher
"FC_PS_PosLesen"	FC 402	FC 402	// PALETTENSPEICHER: Positionen lesen
"FC_PS_WRITE_GUD"	FC 403	FC 403	// PALETTENSPEICHER: Schreibe erweiterte Palettendaten in die GUD-Daten
"FC_PS_JOB_FERTIG"	FC 404	FC 404	// PALETTENSPEICHER: SET/RESET Job fertig
"FC_PS_RS10_SKR"	FC 405	FC 405	// PALETTENSPEICHER: RS10 Rettungsfunktion
"FC_PS_RS10_ABLAUF"	FC 406	FC 406	// PALETTENSPEICHER: RS10 Ablauf
"FC_PS_Hub_Pos"	FC 407	FC 407	// PALETTENSPEICHER: Hub positionieren
"FC408_PS_RESERVE"	FC 408	FC 408	// PALETTENSPEICHER:                                          Reserve
"FC409_PS_RESERVE"	FC 409	FC 409	// PALETTENSPEICHER:                                          Reserve
"FC_HANDLINGSYSTEM_3R"	FC 410	FC 410	// HANDLINGSYSTEM 3R
"FC_HASYST_EROWA"	FC 411	FC 411	// Handlingsystem EROWA/PROMOT
"FC_IF_DMC_ROBOTER"	FC 412	FC 412	// Handlingssystem: Roboterbeladung für Maschinen mit Rüstplatz (Standard)
"FC_DMC_ROB_Beladen"	FC 413	FC 413	// Handlingssystem: Roboter Ablauf Beladen
"FC_DMC_ROB_Entladen"	FC 414	FC 414	// Handlingssystem: Roboter Ablauf Entladen
"FC_ROB_MIT_RPL_MAIN"	FC 415	FC 415	// Handlingssystem: Roboterbeladung für Maschinen mit Rüstplatz (Hauptprogramm)
"FC_ROB_RPL_STAT_ERW"	FC 416	FC 416	// Handlingssystem: Roboter Status-Erweiterung Rüstplatz (BoschRexroth)
"FC_ROB_MPL_STAT_ERW"	FC 417	FC 417	// Handlingssystem: Roboter Status-Erweiterung Maschine (BoschRexroth)
"FC418_FKT_GRP_9"	FC 418	FC 418	// Funktionsgruppe 1                                                    Reserve
"FC419_FKT_GRP_9"	FC 419	FC 419	// Funktionsgruppe 1                                                    Reserve
"FC421_RP_RESERVE"	FC 421	FC 421	// RÜSTPLATZ:                                                             Reserve
"FC422_RP_RESERVE"	FC 422	FC 422	// RÜSTPLATZ:                                                             Reserve
"FC423_RP_RESERVE"	FC 423	FC 423	// RÜSTPLATZ:                                                             Reserve
"FC424_RP_RESERVE"	FC 424	FC 424	// RÜSTPLATZ:                                                             Reserve
"FC425_RP_RESERVE"	FC 425	FC 425	// RÜSTPLATZ:                                                             Reserve
"FC426_RP_RESERVE"	FC 426	FC 426	// RÜSTPLATZ:                                                             Reserve
"FC427_RP_RESERVE"	FC 427	FC 427	// RÜSTPLATZ:                                                             Reserve
"FC428_RP_RESERVE"	FC 428	FC 428	// RÜSTPLATZ:                                                             Reserve
"FC_RPT_ENTRIEGELN"	FC 429	FC 429	// RÜSTPLATZ: Tür entriegeln
"CMM3"	FC 430	FC 430	// Shopmill Nahtstelle Rangierer für Solutionline (Nahtst. entfällt ab SM07.10.06)
"FC_OPERATOR_PANEL"	FC 440	FC 440	// Transfer signals between operator panel and plc-interface
"FC_SMARTKEY_MAIN"	FC 450	FC 450	// Verwaltung von PILZ-Smartkey-Leseeinheit
"FC_SONDER_MAIN"	FC 480	FC 480	// SONDERKONSTRUKTION: Schnittstelle
"FC_SIEM_MCP_STANDARD"	FC 500	FC 500	// SIEMENS Standard Maschinensteuertafel
"FC_SIEM_MCP_OUT"	FC 501	FC 501	// SIEMENS Standard Maschinensteuertafel Ausgänge rangieren
"FC_MASCHTYP_MCP"	FC 509	FC 509	// Maschinentyp -> Maschinensteuertafel
"FC_CI_MAIN"	FC 510	FC 510	// Communication In Main
"FC_CIO_IO_RANGIER"	FC 511	FC 511	// Rangierbaustein Ein- Ausgänge (SOLUTIONLINE)
"FC_DM_MCP"	FC 512	FC 512	// Deckel Maho Maschinensteuertafel Verwaltung
"FC_DM_KONZ_MCP_FC24"	FC 513	FC 513	// Deckel Maho Konzern-Maschinensteuertafel (FC24 aus GP angepasst)
"FC_CI_NCK_PLC"	FC 514	FC 514	// Communication_IN_NCK_PLC
"FC_CO_ERROR"	FC 515	FC 515	// Communication_Out Error
"FC_CO_PLC_NCK"	FC 516	FC 516	// Communication_Out PLC_NCK
"FC_CIO_OEM"	FC 517	FC 517	// OEM: SA Teilenummer Bosch Rexroth
"FC_CO_OEM_Anwahl"	FC 518	FC 518	// OEM: Anwahl der im verwendeten Softkeys
"FC_CO_MAIN"	FC 520	FC 520	// Aufruf Funktionskomponenten am Ende vom Zyklus
"FC540_ACHSE_RESERVE"	FC 540	FC 540	// AX:                                                                 Reserve
"FC_ACHSE_HAUPT"	FC 541	FC 541	// AX: Achssteuerung Haupt einzeln
"FC_ACHSE_HILF"	FC 542	FC 542	// AX: Achssteuerung Hilfs Achse einzeln
"FC543_ACHSE_RESERVE"	FC 543	FC 543	// AX:                                                                 Reserve
"FC_ACHSE_RUND"	FC 544	FC 544	// AX: Rundachse
"FC545_ACHSE_RESERVE"	FC 545	FC 545	// AX:                                                                 Reserve
"FC_ACHSE_RUND_ANFORD"	FC 546	FC 546	// AX: Achsenklemmung Rundachsen
"FC547_ACHSE_RESERVE"	FC 547	FC 547	// AX:                                                                 Reserve
"FC_ACHSE_RPL"	FC 548	FC 548	// AX: Rüstplatz
"FC_ACHSE_RUND_ZUSATZ"	FC 549	FC 549	// AX: Zusatzbaustein Rundachsen
"FC550_SP_RESERVE"	FC 550	FC 550	// Spindel:                                                          Reserve
"FC_ACHSE_SPINDEL"	FC 551	FC 551	// Spindel: im Kanal übergreifende Funktionen
"FC_SP_STERN_DREIECK"	FC 552	FC 552	// Spindel: Stern-Dreieck Umschaltung
"FC_SP_UEBERW"	FC 553	FC 553	// Spindel: Überwachungen
"FC_SP_4STUFEN_GETR"	FC 555	FC 555	// Spindel: 4 Stufiges Getriebe
"FC_SP_UEBERW_DREHZ"	FC 556	FC 556	// Spindel: Drehzahlueberwachung getriebestufenabhaengig
"FC_SP_KOMP_GLAE"	FC 557	FC 557	// Spindel:Glaettungskompensation GMN Spindel
"FC558_SP_RESERVE"	FC 558	FC 558	// Spindel:                                                          Reserve
"FC559_SP_RESERVE"	FC 559	FC 559	// Spindel:                                                          Reserve
"FC_ML_SPI"	FC 560	FC 560	// Minimalmengenschmierung Fa.Vogel
"FC591_DMTDC_RESERVE"	FC 591	FC 591
"FC592_DMTDC_RESERVE"	FC 592	FC 592
"FC593_DMTDC_RESERVE"	FC 593	FC 593
"FC594_DMTDC_RESERVE"	FC 594	FC 594
"FC595_DMTDC_RESERVE"	FC 595	FC 595
"FC_TT_SIMULATION"	FC 600	FC 600	// DM Test-Unterstützung für Maschine IO Simulation
"FC_CONFIG"	FC 700	FC 700	// Maschinen Konfigurations-Daten
"FC_SIEM_DELETE"	FC 723	FC 723	// Siemens IEC Function Blocks:   FC4:   "DELETE"
"FC_SIEM_STRNG_DI"	FC 724	FC 724	// Siemens IEC Function Blocks: FC37: "STRNG_DI"
"FC_AG_LSEND"	FC 1005	FC 1005	// GP-PLC 840D: Daten an den Ethernet-CP senden
"FC_AG_LRECV"	FC 1006	FC 1006	// GP-PLC 840D: Daten von Ethernet-CP empfangen
"FC_AG_LOCK"	FC 1007	FC 1007	// GP-PLC 840D: Datenaustausch mittels FETCH bzw. WRITE sperren
"FC_AG_UNLOCK"	FC 1008	FC 1008	// GP-PLC 840D: Datenaustausch mittels FETCH bzw. WRITE freigeben
"FC_AG_CNTRL"	FC 1010	FC 1010	// GP-PLC 840D: Verbindungen zu diagnostizieren
"MSSTst BA AUTO"	I 0.0	BOOL	// MSST: Taste Betriebsart AUTO_T 21
"MSSTst BA MDA"	I 0.1	BOOL	// MSST: Tate Betriebsart MDA
"MSSTst BA JOG"	I 0.2	BOOL	// MSST: Taste Betriebsart JOG_T 1
"MSSTst Einzelsatz"	I 0.3	BOOL	// MSST: Taste Einzelsatz_T 31
"MSSTst NC-Stop *"	I 0.7	BOOL	// MSST: Taste NC-Stop *_T 41
"MSSTst_NC_Start"	I 1.7	BOOL	// MSST: Taste NC-Start_T 43
"MSSTst 1 INC"	I 2.0	BOOL	// MSST1: Taste 1 INC / MSST2: Taste NC-Stop *
"MSSTst 10 INC"	I 2.1	BOOL	// MSST1: Taste 10 INC / MSST2: Taste NC-Start
"MSSTst 100 INC"	I 2.2	BOOL	// MSST: Taste 100 INC_T 34
"MSSTst 1000 INC"	I 2.3	BOOL	// MSST1: Taste 1000 INC / MSST2: Taste Vorschub Start
"IX_MSST_Ta_2_4"	I 2.4	BOOL	// MSST: Taste Grundstellung fahren
"MSSTst var. INC"	I 2.5	BOOL	// MSST: Inkrement var
"MSSTst Feed Halt *"	I 2.6	BOOL	// MSST: kein Vorschub-Halt
"I_DM_Ta_Feed_Start"	I 2.7	BOOL	// MSST: Taste Vorschub Start_T 47
"I_DM_Ta_Anwahl_WZSp"	I 3.5	BOOL	// MSST: Taste Werkzeugspanner auf zu
"MSSTstReset"	I 3.7	BOOL	// MSST: Taste Reset_T 32
"MSST _T 33"	I 5.7	BOOL	// MSST _T 33  (nicht benutzt)
"MSSTst Handrad EIN"	I 6.2	BOOL	// MSST: Taste Handrad EIN/AUS_T 13 (? Taste zwischen +/-)
"Ta_Foerd_Tuere_entrie"	I 7.7	BOOL	// Taste Tuere entriegeln
"IX_DirektTaste_1_links"	I 8.0	BOOL	// HMI-PRO: OP12/OP15A Direkttaste 1 links
"IX_DirektTaste_2_links"	I 8.1	BOOL	// HMI-PRO: OP12/OP15A Direkttaste 2 links
"IX_DirektTaste_3_links"	I 8.2	BOOL	// HMI-PRO: OP12/OP15A Direkttaste 3 links
"IX_DirektTaste_4_links"	I 8.3	BOOL	// HMI-PRO: OP12/OP15A Direkttaste 4 links
"IX_DirektTaste_5_links"	I 8.4	BOOL	// HMI-PRO: OP12/OP15A Direkttaste 5 links
"IX_DirektTaste_6_links"	I 8.5	BOOL	// HMI-PRO: OP12/OP15A Direkttaste 6 links
"IX_DirektTaste_7_links"	I 8.6	BOOL	// HMI-PRO: OP12/OP15A Direkttaste 7 links
"IX_DirektTaste_8_links"	I 8.7	BOOL	// HMI-PRO: OP12/OP15A Direkttaste 8 links
"IX_DirektTaste_1_rechts"	I 9.0	BOOL	// HMI-PRO: OP12/OP15A Direkttaste 1 rechts
"IX_DirektTaste_2_rechts"	I 9.1	BOOL	// HMI-PRO: OP12/OP15A Direkttaste 2 rechts
"IX_DirektTaste_3_rechts"	I 9.2	BOOL	// HMI-PRO: OP12/OP15A Direkttaste 3 rechts
"IX_DirektTaste_4_rechts"	I 9.3	BOOL	// HMI-PRO: OP12/OP15A Direkttaste 4 rechts
"IX_DirektTaste_5_rechts"	I 9.4	BOOL	// HMI-PRO: OP12/OP15A Direkttaste 5 rechts
"IX_DirektTaste_6_rechts"	I 9.5	BOOL	// HMI-PRO: OP12/OP15A Direkttaste 6 rechts
"IX_DirektTaste_7_rechts"	I 9.6	BOOL	// HMI-PRO: OP12/OP15A Direkttaste 7 rechts
"IX_DirektTaste_8_rechts"	I 9.7	BOOL	// HMI-PRO: OP12/OP15A Direkttaste 8 rechts
"IX_GEN_CABIN_CLOSED"	I 32.0	BOOL	// Kabinentueren geschlossen
"IX_GEN_BUTTON_CONFIRM"	I 32.1	BOOL	// Zustimmungstaste
"IX_SPI_TL_CLP_RELEASED"	I 32.2	BOOL	// Werkzeugspanner geloest
"IX_SPI_TL_CLP_CLAMPED"	I 32.3	BOOL	// Werkzeugspanner gespannt
"IX_HW_SEL"	I 33.1	BOOL	// Aktivierung Handkommandostation
"IX_GEN_OM_2"	I 33.2	BOOL	// Anwahl 2. Betriebsart (kein Einrichten)
"IX_SPI_TL_CLP_SWITCH_REL"	I 33.3	BOOL	// Taster Werkzeugspanner geloest
"IX_CU_MPS_CONTR_CABT_N"	I 34.0	BOOL	// Störung Kuehlmittelanlage Schaltschrank
"IX_GEN_PWR_MODUL_TEMP_OK"	I 34.1	BOOL	// Temperaturüberwachung Versorgungsmodul Antriebe
"IX_GEN_OM_3"	I 34.2	BOOL	// Anwahl 3.Betriebsart
"IX_GEN_OM_4"	I 34.3	BOOL	// Anwahl 4.Betriebsart
"IX_SPI_WYE"	I 35.0	BOOL	// Eingang Sternschaltung
"IX_SPI_DELTA"	I 35.1	BOOL	// Eingang Dreieckschaltung
"IX_GEN_CABIN_LOCKED"	I 35.2	BOOL	// Kabinentueren verriegelt
"IX_GEN_MACHINE_ON"	I 35.3	BOOL	// Rueckmeldung Maschine Ein
"IX_GEN_LUB_PRESSURE_MON"	I 36.0	BOOL	// Druckueberwachung Schmierung Maschine
"IX_GEN_LUB_FILL_LEV_MIN"	I 36.1	BOOL	// Schmierung Maschine: Fuellstand Schmierstoffpumpe
"IX_GEN_HYD_MPS_N"	I 36.2	BOOL	// Störung Hydraulik (Motorschutzschalter/Temperaturüberw
"IX_GEN_HYD_PRESSURE_OK"	I 36.3	BOOL	// Druckueberwachung Hydraulik
"IX_TC_MOTORPROTECTSW_N"	I 37.0	BOOL	// Motorschutzschalter Werkzeugwechsler
"IX_TC_GRP_1_TOOL_MAG"	I 37.1	BOOL	// Werkzeuggreifer 1 Grundstellung Werkzeugmagazin
"IX_TC_GRP_1_SPINDLE"	I 37.2	BOOL	// Werkzeuggreifer 1 Stellung Fraesspindel
"IX_TC_TRANSFERSTATION"	I 37.3	BOOL	// Werkzeugerkennung Uebergabeplatz
"IX_TC_DOOR_CLOSED"	I 38.0	BOOL	// Werkzeugwechsler Tuer geschlossen
"IX_TC_DOOR_OPENED"	I 38.1	BOOL	// Werkzeugwechsler Tuer geoeffnet
"IX_TC_CYL_1_TOOL_MAG"	I 38.2	BOOL	// Pneumatikzylinder 1 Werkzeugmagazin
"IX_TC_CYL_1_HOME_POS"	I 38.3	BOOL	// WW Pneumatikzylinder 1 Grundstellung
"IX_TC_RETENTION_HOME_POS"	I 39.0	BOOL	// Werkzeug-Rueckhalt eingefahren
"IX_TC_RETENTION_MOVD_OU"	I 39.1	BOOL	// Werkzeug-Rueckhalt ausgefahren
"IX_CU_ERROR_TEMP_N"	I 39.7	BOOL	// Kuehlmittelanlage Heiz-/Kuehlgeraet Sammelstoermeldung
"IX_TM_RELEASE"	I 40.0	BOOL	// Schutztuerwaechter Werkzeugbestueckung Werkzeugmagazin
"IX_WM_ZUSTIMMTASTE"	I 40.1	BOOL	// Zustimmtaste Magazin Zweihandbedienung
"IX_WM_Taste_links"	I 40.2	BOOL	// Werkzeugmagazin Linkslauf Handbetaetigung
"IX_WM_Taste_rechts"	I 40.3	BOOL	// Werkzeugmagazin Rechtslauf Handbetaetigung
"IX_CC_MPS_WORM_N"	I 41.1	BOOL	// Motorschutzschalter Spaenefoerderer Schneckenantrieb
"IX_CC_NIVEAU_MAX_N_D"	I 41.2	BOOL	// Diagnose Hebepumpe Spaenefoerderer Not-Aus
"IX_CC_NIVEAU_MAX"	I 41.3	BOOL	// Hebepumpe Spaenefoerderer Not-Aus
"IX_CC_PUMP_ON"	I 43.0	BOOL	// Hebepumpe Spaenefoerderer ein
"IX_CC_PUMP_ON_D"	I 43.1	BOOL	// Diagnose Hebepumpe ein
"IX_CC_PUMP_OFF"	I 43.2	BOOL	// Hebepumpe Spaenefoerderer aus
"IX_CC_PUMP_OFF_D"	I 43.3	BOOL	// Diagnose Hebepumpe aus
"IX_CC_MPS_N"	I 44.0	BOOL	// Motorschutzschalter Spaenefoerderer Kratzerfoerderer
"IX_CC_SWITCH_LEFT"	I 44.1	BOOL	// Spaenefoerderer Linkslauf
"IX_WM_Beladung_zu"	I 44.3	BOOL	// Fenster Werkzeugbestückung geschlossen
"IX_LA_SIGNAL_STAT"	I 45.1	BOOL	// LA: Laser Signal statisch
"IX_LA_RDY"	I 45.2	BOOL	// LA: Laser ok
"IX_LA_MOVED_IN"	I 45.3	BOOL	// LA: Laser eingefahren
"IX_LA_MOVED_OUT"	I 46.0	BOOL	// LA: Laser ausgefahren
"IX_LA_FLAP_CLOSED"	I 46.1	BOOL	// LA: Schmutzblende geschlossen
"IX_OMS_RDY"	I 46.2	BOOL	// Nebel- u.Rauchabscheider betriebsbereit
"IX_OMS_MPS_N"	I 46.3	BOOL	// Motorschutzschalter Nebel- u.Rauchabscheider
"IX_PC_MPL_OCCUPIED"	I 47.0	BOOL	// Palette in der Maschine vorhanden
"IX_PC_MPL_PALLET_RELD"	I 47.1	BOOL	// Palettenklemmung geloest
"IX_PC_MPL_PALLET_CLAMPED"	I 47.2	BOOL	// Palettenklemmung geklemmt
"IX_PC_LIFT_MID"	I 47.3	BOOL	// Palettenwechsler Hub Pos. Mitte
"IX_PC_LIFT_POSITION_4"	I 47.4	BOOL	// Hubeinheit Palettenwechsler Hub schnell
"IX_PC_LIFT_LOWER"	I 48.0	BOOL	// Palettenwechsler Pos. unten
"IX_PC_LIFT_UPPER"	I 48.1	BOOL	// Palettenwechsler Pos. oben
"IX_PC_SST_CHANGE_POS"	I 48.2	BOOL	// Palettenwechsler Ruestplatz Wechselposition
"IX_PC_DOOR_CLOSED"	I 48.3	BOOL	// Kabinentuer Drehpalettenwechsler geschlossen
"IX_PC_SAFETYUNIT_ENABLE"	I 49.0	BOOL	// Freigabe von PNOZ für Palettenwechsler
"IX_MAS_SPANNDRUCK_OK"	I 49.2	BOOL	// Druckschalter Spannvorrichtung gespannt
"IX_PC_SST_CLAMP_PRES_OK"	I 49.3	BOOL	// Spanndruck Ruestplatz vorhanden
"IX_SPI_ROTRA_LUB_PRE_OK"	I 50.0	BOOL	// Druckueberwachung Schmierung M26 (Drehdurchführung)
"IX_SPI_ROTRA_LUB_FILL_OK"	I 50.1	BOOL	// Schmierung M26 (Drehdurchführung) Füllstand
"IX_TL_ML_PRESSURE_OK"	I 50.2	BOOL	// Minimalmengenschmierung Druck ok
"IX_TL_ML_FILL_LEV_OK"	I 50.3	BOOL	// Minimalmengenschmierung Fuellstand ok
"IX_SPI_CLAMPED"	I 51.1	BOOL	// Ueberwachung Fraesspindel geklemmt
"IX_SPI_RELEASED"	I 51.2	BOOL	// Ueberwachung Fraesspindel geloest
"IX_GEN_CAIR_PRESSURE_OK"	I 52.0	BOOL	// Druckueberwachung Druckluft (Systemdruck Pneumatik)
"IX_SPI_LEAK_MONITOR_OK"	I 52.1	BOOL	// Ueberwachung Kuehlmittel SFK
"IX_GEN_GEAR_1_STAGE"	I 52.2	BOOL	// Hauptantrieb 8000 U/min Getriebestellung n<1126 /min
"IX_GEN_GEAR_2_STAGE"	I 52.3	BOOL	// Hauptantrieb 8000 U/min Getriebestellung n>11126 /min
"IX_GEN_OM_BIT_0"	I 53.0	BOOL	// Status Betriebsart
"IX_GEN_OM_BIT_1"	I 53.1	BOOL	// Status Betriebsart
"IX_GEN_OM_BIT_2"	I 53.2	BOOL	// Status Betriebsart
"IX_GEN_OM_BIT_3"	I 53.3	BOOL	// Status Betriebsart
"IX_GEN_EC_TEMP_MONITOR_N"	I 53.4	BOOL	// Schaltschrank Übertemperatur
"IX_CU_MPS_SPI_TR_H_N"	I 54.0	BOOL	// Stoermeldung Kuehlmittelanlage Vorschub Halt
"IX_PC_TABLE_FLUSH_D"	I 54.2	BOOL	// Diagnose Spaenespülung Palettenwechsler
"IX_CU_MOTOR_PAPER_ON"	I 54.3	BOOL	// Motor Papierbandfilter Ein
"IX_KM_NEG_VOR_FUELL"	I 55.0	BOOL	// Kühlmittelanlage Kühlmittelmangel Feinbereich
"IX_KM_NEG_MIN_FUELL"	I 55.2	BOOL	// Fuellstand Feinbereich Minimum
"IX_CU_NIVEAU_MIN"	I 56.0	BOOL	// Kuehlmittel Fuellstand Minimum
"IX_CU_NIVEAU_MIN_D"	I 56.1	BOOL	// Kuehlmittel Diagnose Fuellstand Minimum
"IX_CU_NIVEAU_WAR_MIN"	I 56.2	BOOL	// Kuehlmittel Warnung Fuellstand Minimum
"IX_CU_M7_PRESSURE2_EN"	I 56.3	BOOL	// Kuehlmittel Filterverschmutzung Feinstbereich
"IX_CU_PAPER_END"	I 57.0	BOOL	// Filterband Ende
"IX_D_KM_TPF_PAPIER_ENDE"	I 57.1	BOOL	// Diagnose Filterband Ende
"IX_CU_PAPER_WAR_SHORTAGE"	I 57.2	BOOL	// Warnung Filterband Ende
"IX_D_KM_TPF_PAPIER_WARN"	I 57.3	BOOL	// Diagnose Warnung Filterband Ende
"IX_D_KM_TPF_MOTOR_EIN"	I 58.0	BOOL	// Stoerung Papierbandfilter
"IX_CU_MALFUNCT_N"	I 58.1	BOOL	// keine Stoerung Kuehlmittelanlage
"IX_CU_PAPER_END_A"	I 58.2	BOOL	// Antivalente Ueberwachung Filterband Ende
"IX_CU_PAPER_WAR_SHORT_A"	I 58.3	BOOL	// Antivalente Ueberwachung Papiermangel
"IX_CU_SERVICE"	I 60.3	BOOL	// Filterverschmutzung Feinstbereich Warnung
"IX_KA_NEG_Sammelfehler"	I 62.2	BOOL	// Kuehlaggregat Stoerung
"IX_KA_NEG_Luftfilter"	I 62.3	BOOL	// Kühlaggregat Störmeldung Filterverschmutzung
"IX_TP_CALIBRATION_MOV_OU"	I 64.0	BOOL	// Messeinrichtung Messtaster ausgefahren
"IX_TP_CALIBRATION_MOV_IN"	I 64.1	BOOL	// Messeinrichtung Messtaster eingefahren
"IX_TP_CAL_FLAP_CLSD"	I 64.2	BOOL	// Klappe Messeinrichtung Geschlossen
"IX_MTT_TAB_TEMP_EMSTP"	I 67.0	BOOL	// Temperaturueberwachung Motor Fraes-Drehtisch
"IX_MI_TURNT_TABLE_CLPED"	I 67.1	BOOL	// Klemmung Fraes-Drehtisch geklemmt
"IX_MI_TURNT_TAB_1_RELD"	I 67.2	BOOL	// Klemmung Fraes-Drehtisch geloest
"IX_MI_TURNT_FLC_COOL_N"	I 67.3	BOOL	// Kuehlaggregat Fraes-Drehtisch Durchflusswaechter
"IX_FD_KA_NEG_Luftfilter"	I 68.0	BOOL	// Kuehlaggregat Fraes-Drehtisch Filterverschmutzung
"IX_FD_KA_NEG_Sammelfehle"	I 68.1	BOOL	// Motorschutzschalter Spindelkuehlung
"IX_FD_KA_Temperaturregle"	I 68.2	BOOL	// Kuehlaggregat Fraes-Drehtisch Temperaturregler
"IX_FD_KA_Fuellstand"	I 68.3	BOOL	// Kuehlaggregat Fraes-Drehtisch Fuellstand
"IX_MI_TURNT_PC_CLAMPED"	I 69.0	BOOL	// Palettenklemmung Fraes-Drehtisch geklemmt
"IX_MI_TURNT_PC_RELEASED"	I 69.1	BOOL	// Palettenklemmung Fraes-Drehtisch geloest
"IX_HCD_LUB_PRESSURE_OK"	I 69.3	BOOL	// Druckueberwachung Schmierung Spannfutter
"IX_HCD_LUB_FILL_LEV_OK"	I 70.0	BOOL	// Fuellstand Schmierung Spannfutter
"IX_HCD_SST_UNPRESS"	I 70.1	BOOL	// Ruestplatz Ventil Drucklos
"IX_HCD_SST_FILTER_POLL"	I 70.2	BOOL	// Spannhydraulik Filterverschmutzung Ruestplatz
"IX_HCD_MPL_FILTER_POLL"	I 70.3	BOOL	// Spannhydraulik Filterverschmutzung Maschinenplatz
"IX_PW_RPL_PAL_GEKLEMMT"	I 71.0	BOOL	// Ruestplatz Palettenklemmung geklemmt
"IX_PW_RPL_PAL_GELOEST"	I 71.1	BOOL	// Ruestplatz Palettenklemmung geloest
"IX_HCD_MACHINE_UNLOAD"	I 71.2	BOOL	// Maschine Entladen
"IX_HCD_AXIS_ENABLE"	I 71.3	BOOL	// Freigabe Achsen Sicherheitsschaltgeraet
"IX_SP_SPANN_LOES"	I 72.0	BOOL	// Wahlschalter Spannhydraulik
"IX_SP_AKTIV"	I 72.1	BOOL	// Freigabe Sicherheitsventil
"IX_PC_SST_PALLET_CLAMPED"	I 77.0	BOOL	// G1-36.2  Ruestplatz Palettenklemmung geklemmt
"IX_PC_SST_PALLET_RELD"	I 77.2	BOOL	// G1-36.5  Ruestplatz Palettenklemmung geloest
"IX_TAB_POSITION_0DEG"	I 85.1	BOOL	// Takttisch in Position 0 Grad
"IX_PC_PAL_CAR_UPPER"	I 85.2	BOOL	// Takttisch Palettenträger oben
"IX_PC_PAL_CAR_LOWER"	I 85.3	BOOL	// Takttisch Palettenträger unten
"IX_GEN_T_H_M_FUNCTION"	I 105.0	BOOL	// Freigabe T-H- M-Funktionen
"IX_AL_WARNMELD_PWR_SAG"	I 111.0	BOOL	// Spannungsüberwachung Netz
"IX_TC_TL_CLEAN_MOVED_OUT"	I 111.3	BOOL	// Reinigung Werkzeugkegel ausgefahren
"IX_AL_HYD_FUELL_MAX_OK"	I 112.0	BOOL	// Fuellstand Hydraulik Maximum
"IX_GEN_HYD_FILL_LEV_MIN"	I 112.1	BOOL	// Fuellstand Hydraulik Minimum
"IX_KA_NEG_Stroemungsw"	I 113.1	BOOL	// Kuehlaggregat Stoerung Durchflusswaechter
"IX_KA_NEG_Temp"	I 113.2	BOOL	// Kühlaggregat Stoerung Temperaturregler
"IX_KA_NEG_ND_Fehler"	I 113.3	BOOL	// Kuehlaggregat Stoerung Niederdruckbegrenzung
"IX_KA_NEG_HD_Fehler"	I 114.0	BOOL	// Kuehlaggregat Stoerung Hochdruckbegrenzung
"IX_PC_POSITION_0DEG"	I 114.2	BOOL	// 0 Grad Pos. Palettenwechsler
"IX_PC_POSITION_180DEG"	I 114.3	BOOL	// 180 Grad Pos. Palettenwechsler
"IX_PW_AUF_RP_GESPANNT"	I 114.4	BOOL	// Palettenwechsler Palette auf  Ruestplatz gespannt
"IX_PW_RPL_TUER_2_OFFEN"	I 114.5	BOOL	// Rüstplatz-Tür 2 (rechts) offen
"IX_PW_RPL_TUER_1_OFFEN"	I 114.6	BOOL	// Rüstplatz-Tür 1 (links) offen
"IX_SPI_LUB_FILL_LEV_OK"	I 115.0	BOOL	// Fuellstand Schmierstoffpumpe Oel-Luftschmierung
"IX_SPI_LUB_OIL_PRESS_OK"	I 115.1	BOOL	// Druckueberwachung Schmierung Oel-Luftschmierung
"IX_SPI_LUB_AIR_P_OK"	I 115.2	BOOL	// Druckueberwachung Blasluft Getriebe Hauptantrieb
"IX_OMS_ON_N"	I 115.3	BOOL	// Nebel- u.Rauchabscheider Ein Schalter
"IX_SH_CLAMP_CLAMPED"	I 116.2	BOOL	// Schwenkfraeskopf Klemmung geklemmt
"IX_SH_CLAMP_RELEASED"	I 116.3	BOOL	// Schwenkfraeskopf Klemmung geloest
"IX_PC_LIFT_MID_D"	I 117.2	BOOL	// Palettenwechsler Diagnose Hub Pos. Mitte
"IX_PC_SST_RELEASED"	I 117.3	BOOL	// Ruestplatz Palettenklemmung geloest
"IFX_GEN_EMSTP_CH1_N"	I 120.0	BOOL	// Rueckmeldung Maschine Ein (Kein Not-Aus)
"IX_AL_Tempkomp_TXD"	I 120.1	BOOL	// TEMPERATURKOMPENSATION: Übernahme Temperaturdaten
"IX_TP_BATTERIE_MIN"	I 120.2	BOOL	// Messtaster Batteriewarnung
"IX_TP_RDY"	I 120.3	BOOL	// Messtaster Betriebsbereit
"IFX_GEN_OM1_CH1_SEL"	I 121.0	BOOL	// Freigabe Drehzahl Maximum (Betriebsart 1)
"IFX_GEN_OM2_CH1_SEL"	I 121.1	BOOL	// Freigabe Betriebsart 2
"IFX_GEN_OM3_4_CH1_SEL"	I 121.2	BOOL	// Freigabe Betriebsart 3/4
"IX_HR_plus_Taste"	I 121.3	BOOL	// Handrad Taste +
"IX_HR_minus_Taste"	I 122.0	BOOL	// Handrad Taste -
"IX_HR_Eilgang_Taste"	I 122.1	BOOL	// Handrad Taste Eilgang
"IX_HR_FKT_Taste_F1"	I 122.2	BOOL	// Handrad Taste F1
"IX_HR_FKT_Taste_F2"	I 122.3	BOOL	// Handrad Taste F2
"IX_HR_FKT_Taste_F3"	I 123.0	BOOL	// Handrad Taste F3
"IX_HR_Achsanwahl_Bit_0"	I 123.1	BOOL	// GRAY-Code Achsumschaltung Bit 0
"IX_HR_Achsanwahl_Bit_1"	I 123.2	BOOL	// GRAY-Code Achsumschaltung Bit 1
"IX_HR_Achsanwahl_Bit_2"	I 123.3	BOOL	// GRAY-Code Achsumschaltung Bit 2
"IX_WM_WZ_einlegen"	I 125.0	BOOL	// Quittierung Werkzeug einlegen
"IX_WM_WZ_entnehmen"	I 125.1	BOOL	// Quittierung Werkzeug entnehmen
"IX_SPI_FEED_STOP_N"	I 126.0	BOOL	// Spindel/Vorschub Halt
"IX_PS_SST_DOOR_FRONT_LKD"	I 144.0	BOOL	// Ruestplatztuer Palettenspeichersystem verriegelt vorn
"IX_PS_SST_DOOR_REAR_LKD"	I 144.1	BOOL	// Ruestplatztuer Palettenspeichersystem verriegelt hinten
"IX_PS_SST_DOOR_FRT_CLSD"	I 144.2	BOOL	// Ruestplatztuer vorn geschlossen
"IX_PS_SST_DOOR_REAR_CLSD"	I 144.3	BOOL	// Ruestplatztuer hinten geschlossen
"IX_D_PS_RPL_PAL_VORH"	I 145.0	BOOL	// Palette Ruestplatz vorhanden Diagnose
"IX_PS_SST_OCCUPIED"	I 145.1	BOOL	// Palette Ruestplatz vorhanden
"IX_PS_SST_HOME_POS"	I 145.2	BOOL	// Ruestplatz Palettenspeichersystem Grundstellung
"IX_PS_LIFT_DOOR_CLOSED"	I 145.3	BOOL	// Hubtuere Palettenwechsel Sicherheitsschalter
"IX_PS_TURN_STATION_OCC"	I 146.0	BOOL	// Palette auf Schlitten vorhanden Drehachse
"IX_PS_STO_ST_PAL_EXI"	I 146.1	BOOL	// Ueberwachung Palette vorhanden Ablageplatz
"IX_PS_STO_ST_PAL_EXI_A"	I 146.2	BOOL	// Ueberwachung Palette vorhanden Ablageplatz Öffner
"IX_PS_ROTARY_REG_OK"	I 146.3	BOOL	// Meldung Drehbereichsbegrenzung betaetigt
"IX_PS_TURN_ST_LIFT_LOW"	I 147.0	BOOL	// Sensor Dreheinheit unten
"IX_PS_TURN_ST_LIFT_UPP"	I 147.1	BOOL	// Sensor Dreheinheit oben
"IX_PS_FRG_AR_PSACHS"	I 148.0	BOOL	// Antriebsfreigabe Arbeitsraum Palettenspeichersystem
"IX_PS_FRG_AR_NCRPL"	I 148.1	BOOL	// Antriebsfreigabe Arbeitsraum Rüstplatz
"IX_PS_EMERG_STOP_N"	I 148.2	BOOL	// Rueckmeldung Not-Aus Palettenspeichersystem
"IX_PS_SAFETYUNIT_READY"	I 148.3	BOOL	// PNOZmulti Palettenspeichersystem betriebsbereit
"IX_MI_TURNT_TAB_CLPED_D"	I 150.2	BOOL	// Diagnose Klemmung geklemmt
"IX_MI_TURNT_TABLE_RELD_D"	I 150.3	BOOL	// Diagnose Klemmung geloest
"IX_MI_TURNT_LUB_FILL_OK"	I 152.0	BOOL	// Fuellstand Schmierstoffpumpe Fraes-Drehtisch
"IX_MI_TURNT_C_PULS_LUB"	I 152.1	BOOL	// Zyklenschalter Progressievverteiler
"IX_CA_FLOW_CONTROL_SPI_N"	I 153.0	BOOL	// Durchflusswaechter Kuehlkreislauf Hauptantrieb
"IX_KA_N_ACHS_DURCHFLUSSW"	I 153.1	BOOL	// Durchflusswaechter Kuehlkreislauf Vorschubantriebe
"IX_FD_N_DURCHFL_LAGER"	I 153.2	BOOL	// Durchflusswaechter Kuehlkreislauf Lager FD-Tisch
"IX_MI_TURNT_FLC_STA_N"	I 153.3	BOOL	// Durchflusswaechter Kuehlkreislauf Stator FD-Tisch
"IX_U_AXIS_ALM_CDE_BIT_0"	I 172.0	BOOL	// U-Achse Alarm Bit 0
"IX_U_AXIS_ALM_CDE_BIT_1"	I 172.1	BOOL	// U-Achse Alarm Bit 1
"IX_U_AXIS_ALM_CDE_BIT_2"	I 172.2	BOOL	// U-Achse Alarm Bit 2
"IX_U_AXIS_ALM_CDE_BIT_3"	I 172.3	BOOL	// U-Achse Alarm Bit 3
"IX_U_AXIS_CONFIRM"	I 173.0	BOOL	// U-Achse Quittierung
"IX_U_AXIS_ALARM_N"	I 173.1	BOOL	// U-Achse kein Alarm
"IX_U_AXIS_TOOL_ACTIVE_N"	I 173.2	BOOL	// U-Achse keine Bearbeitung
"IX_U_AXIS_TOOL_READY"	I 173.3	BOOL	// U-Achse Werkzeug Betriebsbereit
"IX_U_AXIS_REF_SIGNAL"	I 174.0	BOOL	// U-Achse Referenzimpuls
"IX_U_AXIS_READY"	I 174.1	BOOL	// U-Achse Achse Betriebsbereit
"IX_U_AXIS_SWITCH_PLUS"	I 174.2	BOOL	// U-Achse Endschalter positiv
"IX_U_AXIS_SWITCH_MINUS"	I 174.3	BOOL	// U-Achse Endschalter negativ
"IX_GEN_HYD_TEMP_OK"	I 500.0	BOOL	// Temperaturueberwachung Hydraulik
"IX_TC_CYL_1_SPINDLE"	I 1000.0	BOOL	// Werkzeugmagazin Stellung Spindel
"IX_TM_TOOL_CYL_LOCKED"	I 1000.1	BOOL	// Pneumatikzylinder Werkzeug loesen eingefahren Grundstellung
"IX_TM_TOOL_CYL_UNLOCKED"	I 1000.2	BOOL	// Pneumatikzylinder Werkzeug loesen ausgefahren
"IX_TM_TOOL_SPI_LOCKED"	I 1000.3	BOOL	// Werkzeug verriegelt Wechselposition
"IX_WM_WZ_MAN_Relase"	I 1000.4	BOOL	// Werkzeug manuell entriegeln
"IX_TM_TOOL_MAN_CLAMP"	I 1000.5	BOOL	// Werkzeug manuell klemmen
"IX_CU_NIVEAU_MAX"	I 1000.6	BOOL	// Kuehlmittel Fuellstand Maximum
"IX_CU_SAFETY_EMSTP_EN"	I 1000.7	BOOL	// Freigabe Kuehlmittelanlage PNOZ Not-Aus
"IX_CU_SAFETYUNIT_CAB_EN"	I 1001.0	BOOL	// Freigabe Kuehlmittelanlage PNOZ Kabinentuer geschlossen
"IX_PW_QUIT_Freigabe"	I 1001.1	BOOL	// Quittierung Freigabe Palettenwechsler
"IX_TM_TOOL_SST_LOCKED"	I 1001.2	BOOL	// Werkzeug verriegelt Werkzeugeingabestation
"IX_TM_TOOL_MAN_RELEASE"	I 1001.4	BOOL	// Werkzeug manuell loesen
"IX_TM_TST_OCC"	I 1001.5	BOOL	// Uebergabeplatz belegt vertikale Kette ohne TPU
"IX_GEN_AXIS_SPEED_RPM_OK"	I 1002.0	BOOL	// Ueberwachung Drehzahlbegrenzung
"IX_GEN_AXIS5_CLAMPED"	I 1002.1	BOOL	// Klemmung 4.Achse geklemmt
"IX_PC_LIFT_POSITION_1"	I 1002.2	BOOL	// Palettenwechsler Hub Position 1
"IX_PC_LIFT_POSITION_2"	I 1002.3	BOOL	// Palettenwechsler Hub Position 2
"IX_PC_LIFT_POSITION_3"	I 1002.4	BOOL	// Palettenwechsler Hub Position 3
"IX_SP_HYD_EIN"	I 1002.5	BOOL	// Bereichsschalter Spannhydraulik Ein
"IX_SP_HYD_FUEL_OK"	I 1002.6	BOOL	// Spannhydraulik Ueberwachung Fuellstand
"IX_SP_HYD_NEG_STOERUNG"	I 1002.7	BOOL	// Spannhydraulik Motorschutzschalter ok
"IX_SP_HYD_RPL_LOESEN"	I 1003.0	BOOL	// Fußschalter Spannhydraulik entspannen
"IX_SP_HYD_RPL_SPANNEN"	I 1003.1	BOOL	// Fußschalter Spannhydraulik spannen
"IX_SP_HYD_TEMP_OK"	I 1003.2	BOOL	// Spannhydraulik Temperatur ok
"IX_KM_DRUCK2_M7_EIN"	I 1003.3	BOOL	// Kuehlmittel Freigabe Maschine Druckstufe 2
"IX_KM_DRUCK0_M7_EIN"	I 1004.0	BOOL	// Kuehlmittel Freigabe Maschine Druckstufe 0
"IX_PC_TST_OCC"	I 1004.1	BOOL	// Palette auf PW-Übergabeplatz vorhanden (bei Palettenspeicher)
"IX_KM_FEINB_MIN"	I 1004.3	BOOL	// Feinbereich Fuellstand Minimum
"IX_KM_KRATZER_EIN"	I 1004.4	BOOL	// Feinbereich Fuellstand Regeneration
"IX_D_KM_KRATZER_EIN"	I 1004.5	BOOL	// Diagnose Feinbereich Regeneration
"IX_D_KM_FEINB_MIN"	I 1004.6	BOOL	// Diagnose Feinbereich Minimum
"IX_CU_MOTOR_PAPER_ON_A"	I 1004.7	BOOL	// Kuehlmittel Diagnose Fuellstand Filtermulde
"IX_CU_NIVEAU_MIN_MAX_D"	I 1005.0	BOOL	// Kuehlmittel Diagnose Niveaukontrolle Feinbereich
"IX_D_KM_VOR_MIN_NIVEAU"	I 1005.1	BOOL	// Kuehlmittel Diagnose Vorwarnung Feinbereich
"IX_TC_CYL_1_ENABLE"	I 1005.3	BOOL	// Freigabe drehen Werkzeugmagazin
"IX_CA2_WARNMSG_N"	I 1005.4	BOOL	// Kuehlaggregat 2 Warnmeldung
"IX_CA2_MALFUNCT_2_N"	I 1005.5	BOOL	// Kuehlaggregat 2 Störmeldung Prioritaet 2
"IX_CA2_MALFUNCT_1_N"	I 1005.6	BOOL	// Kuehlaggregat 2 Störmeldung Prioritaet 1
"IX_KM_WARN_KSS_TEMP"	I 1005.7	BOOL	// Kuehlmittel Warnung Temperaturueberwachung
"IX_KM_NEG_FEHLER_TEMP"	I 1006.0	BOOL	// Sammelstoermeldung Kuehl/Heizaggregat Kuehlmittelanlage
"IX_TC_POSITION_ENABLE_TM"	I 1006.1	BOOL	// Werkzeugwechsler Position Freigabe Werkzeugmagazin
"IX_TM_PLACE_OCCUPIED"	I 1006.2	BOOL	// Magazinplatz belegt
"IX_TM_TLOAD_WDOW_CLOSE"	I 1006.3	BOOL	// Fenster Rüstplatz geschlossen
"IX_TM_TLOAD_APPROVAL"	I 1006.4	BOOL	// Zustimmtaste Rüstplatz
"IX_TM_TLOAD_ACK_TOOL_IN"	I 1006.5	BOOL	// Bestätigung Werkzeug einlegen
"IX_TM_TLOAD_ACK_TOOL_OUT"	I 1006.6	BOOL	// Bestätigung Werkzeug entnommen
"IX_TM_TLOAD_CHAIN_PLUS"	I 1006.7	BOOL	// Taste Kettenmagazin Plus-Richtung (rechts) fahren
"IX_TM_TLOAD_CHAIN_MINUS"	I 1007.0	BOOL	// Taste Kettenmagazin Minus-Richtung (links) fahren
"IX_KM_SPRUEHPIST_RPL_EIN"	I 1009.0	BOOL	// Anforderung Spülpistole Rüstplatz Ein
"IX_SST_ENABLE_ROTATE"	I 1009.1	BOOL	// Antriebsfreigabe Ruestplatz
"IX_SST_LEFT_ROTATE"	I 1009.2	BOOL	// Ruestplatz drehen Links
"IX_SST_RIGHT_ROTATE"	I 1009.3	BOOL	// Ruestplatz drehen Rechts
"IX_SST_CONFIRM"	I 1009.4	BOOL	// Zustimmungstaste NC-Ruestplatz drehen
"IX_GEN_DRIVES_ENABLE"	I 1010.0	BOOL	// Vorschubfreigabe X/Y/Z-Achse 4./5.-Achse
"IX_GEN_READ_IN_ENABLE"	I 1010.1	BOOL	// Einlesefreigabe
"IX_TC_ENABLE"	I 1010.2	BOOL	// Freigabe Werkzeugwechsler
"IX_PC_ENABLE"	I 1010.3	BOOL	// Freigabe Drehpalettenwechsler
"IX_SH_ENABLE"	I 1010.4	BOOL	// Freigabe Schwenkfrässkopf
"IX_CA_MPS_N"	I 1010.5	BOOL	// Motorschutzschalter Luefter Waermetauscher Kuehlaggregat
"IX_TM_COUNT_PULS"	I 1010.6	BOOL	// Zaehlimpuls Werkzeugmagazin
"IX_TM_REF_SIGNAL"	I 1010.7	BOOL	// Referenzimpuls Werkzeugmagazin
"IX_CC_AUTO"	I 1011.0	BOOL	// Spaenefoerderer Betriebsart Automatik
"IX_CC_SWITCH_RIGHT"	I 1011.1	BOOL	// Spaenefoerderer Rechtslauf
"IX_LA_SIGNAL_DYN"	I 1011.2	BOOL	// LA: Laser Signal dynamisch
"IX_MAS_NEG_SPANNDRUCK"	I 1011.4	BOOL	// Druckschalter Spannvorrichtung geloest
"IX_GEN_AXIS4_CLP_RELEASE"	I 1011.5	BOOL	// Klemmung 4.Achse auf
"IX_AL_4ACHS_KLE_geloest"	I 1011.6	BOOL	// Klemmung 4.Achse gelöst
"IX_GEN_AXIS4_CLAMP"	I 1011.7	BOOL	// Klemmung 4.Achse zu
"IX_GEN_AXIS5_CLP_RELD"	I 1012.0	BOOL	// Klemmung 5.Achse gelöst
"IX_WM_TAS_Beladung_auf"	I 1012.1	BOOL	// Freigabe Magnetverriegelung WZB (Fenster Werkzeugbestückung) oeffnen
"IX_WM_TAS_Beladung_zu"	I 1012.2	BOOL	// Freigabe Magnetverriegelung WZB-geschlossen
"IX_WM_Beladung_auf"	I 1012.3	BOOL	// Werkzeugbestueckung Fenster geoffnet
"IX_WM_1_Eingabeplatz"	I 1012.4	BOOL	// Ueberwachung Werkzeugbestueckung Platz 1
"IX_TC_TL_CLEAN_HOME_POS"	I 1012.5	BOOL	// Reinigung Werkzeugkegel eingefahren
"IX_KA_NEG_Wasserstand"	I 1012.6	BOOL	// Kuehlaggregat Stoerung Fuellstand
"IX_TM_MONITOR_SWITCH"	I 1012.7	BOOL	// Umschaltung Werkzeugeingabefunktion
"IX_SH_POSITION_HORZ"	I 1013.0	BOOL	// Stellung Schwenkfraeskopf waagrecht
"IX_SH_POSITION_VERT"	I 1013.1	BOOL	// Stellung Schwenkfraeskopf senkrecht
"IX_WM_2_Eingabeplatz"	I 1013.2	BOOL	// Ueberwachung Werkzeugbestueckung Platz 2
"IX_WM_3_Eingabeplatz"	I 1013.3	BOOL	// Ueberwachung Werkzeugbestueckung Platz 3
"IX_WM_4_Eingabeplatz"	I 1013.4	BOOL	// Ueberwachung Werkzeugbestueckung Platz 4
"IX_WW_Ablageplatz"	I 1013.5	BOOL	// Ueberwachung Ablageplatz Handlingsystem
"IX_D_WW_Ablageplatz"	I 1013.6	BOOL	// Diagnose Ueberwachung Ablageplatz
"IX_WM_TOPF_SPA_OFFEN"	I 1013.7	BOOL	// Pneumatikzylinder Werkzeugspanner geoeffnet
"IX_WM_TOPF_SPA_ZU_MIT_WZ"	I 1014.0	BOOL	// Pneumatikzylinder Werkzeugspanner geschlossen mit Werkzeug
"IX_WM_TOPF_SPA_ZU_O_WZ"	I 1014.1	BOOL	// Pneumatikzylinder Werkzeugspanner geschlossen ohne Werkzeug
"IX_GEN_SAFETYUNIT_RDY"	I 1014.2	BOOL	// Betriebsbereit Sicherheitsschaltgeraet
"IX_DH_CLAMP_RELEASED"	I 1014.3	BOOL	// Klemmung geloest NC-Teilapparat
"IX_WK_SPINDEL_ABDECKUNG"	I 1014.4	BOOL	// Spindel Abdeckung geschlossen
"IX_CU_SUP_F_REG_OFF_D"	I 1015.0	BOOL	// Kuehlmittel Diagnose Feinstbereich Maximum
"IX_CU_SUP_F_REG_ON_D"	I 1015.1	BOOL	// Kuehlmittel Diagnose Feinstbereich Minimum
"IX_CU_SUP_F_REG_MIN_D"	I 1015.2	BOOL	// Kuehlmittel Diagnose Feinstbereich Grenzwertmeldung
"IX_CU_SUP_F_REG_OFF"	I 1015.3	BOOL	// Kuehlmittel Feinstbereich Fuellstand Maximum
"IX_CU_SUP_F_REG_ON"	I 1015.4	BOOL	// Kuehlmittel Feinstbereich Fuellstand Minimum -> Pumpe Ein
"IX_CU_SUP_F_REG_MIN"	I 1015.5	BOOL	// Kuehlmittel Feinstbereich Fuellstand Grenzwertmeldung
"IX_CU_NIVEAU_MIN_MAX"	I 1015.6	BOOL	// Kuehlmittel Niveaukontrolle Feinbereich
"IX_KM_VOR_MIN_NIVEAU"	I 1015.7	BOOL	// Kuehlmittel Vorwarnung Feinbereich Minimum
"IX_SP_MPL_ENTKUPPELT"	I 1016.0	BOOL	// Spannhydraulik Maschinenplatz entkuppelt
"IX_SP_MPL_GEKUPPELT"	I 1016.1	BOOL	// Spannhydraulik Maschinenplatz gekuppelt
"IX_SP_RPL_ENTKUPPELT"	I 1016.2	BOOL	// Spannhydraulik Rüstplatz entkuppelt
"IX_SP_RPL_GEKUPPELT"	I 1016.3	BOOL	// Spannhydraulik Rüstplatz gekuppelt
"IX_AL_SICHERUNG_230V_OK"	I 1016.6	BOOL	// Diagnose Sicherung 230V
"IX_AL_Sicherung_24V_OK"	I 1016.7	BOOL	// Diagnose Sicherung 24V
"IX_KM_SF_KRATZ_NIV_MAX"	I 1017.0	BOOL	// Max. Niveau-Überwachung  Kratzerförderer
"IX_D_KM_SF_KRATZ_NIV_MAX"	I 1017.1	BOOL	// Diagnose Max. Niveau-Überwachung  Kratzerförderer
"IX_KM_SF_PUMPE_EIN"	I 1017.2	BOOL	// Niveaukontrolle Schmutztank Hebepumpe „Ein“
"IX_D_KM_SF_NEG_PUMPE_EIN"	I 1017.3	BOOL	// Diagnose Niveau Schmutztank Hebepumpe „Ein“
"IX_KM_SF_PUMPE_AUS"	I 1017.4	BOOL	// Niveaukontrolle Schmutztank Hebepumpe „Aus“
"IX_D_KM_SF_NEG_PUMPE_AUS"	I 1017.5	BOOL	// Diagnose Niveau Schmutztank Hebepumpe „Aus“
"IX_KM_SF_TANK_NIV_MAX"	I 1017.6	BOOL	// Maximale Niveaukontrolle Schmutztank
"IX_D_KM_SF_NEG_TANK_MAX"	I 1017.7	BOOL	// Diagnose Maximale Niveaukontrolle Schmutztank
"IX_TT_ausgeschwenkt"	I 1018.0	BOOL	// Messtaster Tisch TS27R ausgeschwenkt
"IX_TT_eingeschwenkt"	I 1018.1	BOOL	// Messtaster Tisch TS27R eingeschwenkt
"IX_SPI_IAS_MONITOR"	I 1018.2	BOOL	// C1-13.4 Durchflusswaechter Kuehlmittel 2 (M7)
"IX_SPI_FLOW_CONTROL_MON"	I 1018.3	BOOL	// C1-13.7 Durchflusswaechter Leitungsueberwachung (M7)
"IX_KM_FILTER_FEINB_OK"	I 1018.4	BOOL	// B3-90.3 Filter Feinst-Bereich OK
"IX_PC_SRT_LIFT_2_MID"	I 1020.0	BOOL	// Palettenwechsler Position vor Mitte
"IX_PC_SRT_LIFT_2_LOW"	I 1020.1	BOOL	// Palettenwechsler Position vor unten
"IX_PC_LIFT_POSITION_2_D"	I 1020.2	BOOL	// Palettenwechsler Diagnose Position 2
"IX_MI_TURNT_TAB_2_RELD"	I 1021.0	BOOL	// Klemmung Fraes-Drehtisch geloest Naeherungsschalter
"IX_TM_TPU_GET_TOOL"	I 1022.0	BOOL	// Transporteinheit ist auf Werkzeugkegel gefahren
"IX_TM_TPU_RELEASE_TOOL"	I 1022.1	BOOL	// Transporteinheit ist vom Werkzeugkegel weggefahren
"IX_TM_TPU_TRANSFERPOS"	I 1022.2	BOOL	// Transporteinheit ist zur Übergabeposition gefahren
"IX_TM_TPU_MAGAZINPOS"	I 1022.3	BOOL	// Transporteinheit ist zur Magazinposition gefahren
"IX_TM_MAG_TOOL_UNLOCK"	I 1022.4	BOOL	// Werkzeug an Magazinposition ist entriegelt
"IX_TM_MAG_TOOL_LOCK"	I 1022.5	BOOL	// Werkzeug an Magazinposition ist verriegelt
"IX_TM_TLOAD_TOOL_UNLOCK"	I 1022.6	BOOL	// Werkzeug am Rüstplatz ist entriegelt
"IX_TM_TLOAD_TOOL_LOCK"	I 1022.7	BOOL	// Werkzeug am Rüstplatz ist verriegelt
"IX_TM_TLOAD_PIN_LOCK"	I 1023.0	BOOL	// Werkzeug am Rüsplatz entriegeln
"IX_TM_MAG_PIN_LOCK"	I 1023.1	BOOL	// Verriegelungspin Magazinposition verriegelt
"IX_TM_TLOAD_TOOL_INSERT"	I 1023.2	BOOL	// Positionsüberwachung Werkzeug Rüstplatz
"IX_SP_RPL_SPST1_ANWAHL"	I 1024.0	BOOL	// Spannhydraulik Taster Spannstelle 1
"IX_SP_RPL_SPST2_ANWAHL"	I 1024.1	BOOL	// Spannhydraulik Taster Spannstelle 2
"IX_SP_RPL_SPST3_ANWAHL"	I 1024.2	BOOL	// Spannhydraulik Taster Spannstelle 3
"IX_SP_RPL_SPST4_ANWAHL"	I 1024.3	BOOL	// Spannhydraulik Taster Spannstelle 4
"IX_SP_AUFL_ST1_GESPANNT"	I 1024.4	BOOL	// Kontrolle Auflage Spannstelle 1 gespannt ok
"IX_SP_AUFL_ST2_GESPANNT"	I 1024.5	BOOL	// Kontrolle Auflage Spannstelle 2 gespannt ok
"IX_SP_AUFL_ST3_GESPANNT"	I 1024.6	BOOL	// Kontrolle Auflage Spannstelle 3 gespannt ok
"IX_SP_AUFL_ST4_GESPANNT"	I 1024.7	BOOL	// Kontrolle Auflage Spannstelle 4 gespannt ok
"IX_TOOL_CLAMP_CLPD_WO_TL"	I 1025.0	BOOL	// Werkzeugspanner gespannt ohne Werkzeug
"IX_WK_ZYL_1_GST"	I 1025.1	BOOL	// Werkzeugtraeger Zylinder 1 Grundstellung
"IX_WK_ZYL_1_WE_POS"	I 1025.2	BOOL	// Werkzeugtraeger Zylinder 1 Wechselposition
"IX_WK_ZYL_2_GST"	I 1025.3	BOOL	// Werkzeugtraeger Zylinder 2 Grundstellung
"IX_WK_ZYL_2_WE_POS"	I 1025.4	BOOL	// Werkzeugtraeger Zylinder 2 Wechselposition
"IX_WK_KLAPPE_AUF"	I 1025.5	BOOL	// Werkzeugklappe geoffnet
"IX_WK_KLAPPE_ZU"	I 1025.6	BOOL	// Werkzeugklappe geschlossen
"IX_WK_WZ_1_VORHANDEN"	I 1025.7	BOOL	// Winkelfraeskopf 1 vorhanden
"IX_WK_WZ_2_VORHANDEN"	I 1026.0	BOOL	// Winkelfraeskopf 2 vorhanden
"IX_FMS_OM_DISABLED"	I 1027.0	BOOL	// Schluesselschalter Deaktivierung Uebergabeplatz/ Maschine/Palettenspeichersystem
"IX_ROBOT_AUTO"	I 1028.0	BOOL	// Betriebsart Automatik Handlingsystem
"IX_ROBOT_LOAD_END"	I 1028.1	BOOL	// Handlingsystem Rueckmeldung Werkstueckwechsel
"IX_ROBOT_CHUCKS_CLOSED"	I 1028.2	BOOL	// Spannfutter gespannt
"IX_ROBOT_DOOR_CLOSED"	I 1028.3	BOOL	// Hubtuer Werkstuecklader geschlossen
"IX_ROBOT_DOOR_OPENED"	I 1028.4	BOOL	// Hubtuere Werkstuecklader offen
"IX_ROBOT_NEG_ERROR"	I 1028.5	BOOL	// Fehler Handlingsystem
"IX_ROBOT_NEUTRAL"	I 1028.6	BOOL	// Grundstellung Handlingsystem
"IX_WA_ENABLE_DOOR_OPEN"	I 1028.7	BOOL	// Freigabe Kabinentüre entriegeln
"IX_CU_M7_PRESSURE0_EN"	I 1030.0	BOOL
"IX_CU_M7_PRESSURE1_ON"	I 1030.1	BOOL
"IX_CU_SAVETY_EMSTP_EN"	I 1030.2	BOOL
"IX_CU_SAVETYUNIT_CAB_EN"	I 1030.3	BOOL
"IX_GEN_OM_SERVICE_ACTIVE"	I 1030.4	BOOL
"IX_VMS_BEARING_ERROR"	I 1030.5	BOOL
"IX_VMS_BEARING_WAR"	I 1030.6	BOOL
"IX_VMS_CRASH"	I 1030.7	BOOL
"IX_VMS_MEASURING_BEA_RDY"	I 1031.0	BOOL
"IX_VMS_UNBALANCE_ERROR"	I 1031.1	BOOL
"IX_VMS_UNBALANCE_WAR"	I 1031.2	BOOL
"IX_VMS_VIBRATION_FAULT_D"	I 1031.3	BOOL
"IX_CU_M7_PRESSURE1_EN"	I 1031.4	BOOL	// M-EINGANG: KM Druck 1 M7 Freigabe
"IX_RELEASEUNI_GET_TOOL"	I 1032.0	BOOL	// Ausrückstation Position Werkzeugkegel
"IX_RELEASEUNI_RELEASE_T"	I 1032.1	BOOL	// Ausrückstation Position Grundstellung
"IX_RELEASEUNI_TRANSPOS"	I 1032.2	BOOL	// Ausrückstation Position Übergabeposition
"IX_RELEASEUNI_MAGAZINPOS"	I 1032.3	BOOL	// Ausrückstation Position Magazinposition
"IX_RELU_MAG_TOOL_UNLKD"	I 1032.4	BOOL	// Ausrückstation Werkzeug im Greifer gelöst
"IX_RELU_MAG_TOOL_LKD"	I 1032.5	BOOL	// Ausrückstation Werkzeug im Greifer gespannt
"IX_RELU_MAG_PIN_LKD"	I 1032.6	BOOL	// Ausrückstation Verriegelungspin Magazinplatz verriegelt
"IX_RELEASEUNI_MAG_OCC"	I 1032.7	BOOL	// Ausrückstation Magazinplatz belegt
"IX_RELU_TST_TOOL_UNLKD"	I 1033.0	BOOL	// Ausrückstation Kettenverriegelungszylinder ausgefahren
"IX_RELEASEUNI_TST_OCC"	I 1033.1	BOOL	// Ausrückstation Übergabeplatz belegt
"IX_RELU_TST_TOOL_LKD"	I 1033.2	BOOL	// Ausrückstation Kettenverriegelungszylinder eingefahren
"IX_TC_MAGAZINPOS"	I 1033.4	BOOL
"IX_TC_SPIPOS"	I 1033.5	BOOL
"IX_CA_WARNMSG_N"	I 1040.0	BOOL	// Kuehlaggregat Warnmeldung (Filterverschmutzung)
"IX_CA_MALFUNCT_1_N"	I 1040.1	BOOL	// Kuehlaggregat Störmeldung Prioritaet 1
"IX_CA_MALFUNCT_2_N"	I 1040.2	BOOL	// Kuehlaggregat Störmeldung Prioritaet 2
"IX_PC_LUB_FILL_LEV_OK"	I 1052.0	BOOL	// Schmierung Palettenwechsler Überwachung Füllstand
"IX_PC_LUB_PRESSURE_OK"	I 1052.1	BOOL	// Schmierung Palettenwechsler Drucküberwachung
"IX_CU_NIVEAU_WAR_MIN_D"	I 1056.1	BOOL	// Kuehlmittel Diagnose Warnung Minimum
"IX_CU_NIVEAU_MAX_D"	I 1057.1	BOOL	// Kuehlmittel Diagnose Fuellstand Maximum
"IX_SO_WFK_ANGEDOCKT"	I 1057.2	BOOL	// Wiegenfräskopf angedockt / Klemmposition erreicht
"IX_SO_WFK_KLE_GEKLEMMT"	I 1057.3	BOOL	// Wiegenfräskopf Klemmung geklemmt
"IX_SO_WFK_KLE_GELOEST"	I 1057.4	BOOL	// Wiegenfräskopf Klemmung gelöst
"IX_SO_DMS_UEBERWACH_OEL"	I 1057.5	BOOL	// Drehmomentstütze Ölstandsüberwachung Niveau
"IX_HCD_MALFUNCT_N"	I 1062.0	BOOL	// Spannhydraulik Betriebsbereit   /H4-09.2
"IX_HCD_FILL_LEV_OK"	I 1062.1	BOOL	// Spannhydraulik Ueberwachung Fuellstand   /H4-20.7
"IX_HCD_TEMP_OK"	I 1062.2	BOOL	// Spannhydraulik Temperaturueberwachung   /H4-20.6
"IX_HCD_ON"	I 1062.3	BOOL	// Bereichsschalter Spannhydraulik Ein   /H4-09.4
"IX_PC_CONFIRM_ENABLE"	I 1062.5	BOOL	// Quittierung Freigabe Palettenwechsler   /G1-05.3
"IX_HCD_SST_CLAMP"	I 1062.6	BOOL	// Spannhydraulik Spannvorrichtung Spannen   /H4-10.2
"IX_HCD_SST_RELEASE"	I 1062.7	BOOL	// Spannhydraulik Spannvorrichtung loesen   /H4-10.5
"IX_HCD_SST_ENGAGED"	I 1067.4	BOOL	// Hydraulik Rüstplatz Kupplung angekuppelt   /H4-07.7
"IX_HCD_SST_DISENGAGED"	I 1067.5	BOOL	// Hydraulik Rüstplatz Kupplung abgekuppelt   /H4-07.7
"IX_HCD_SST_CLA_POI_1_SEL"	I 1078.4	BOOL	// Spannhydraulik Anwahl Spannkreis 1   /H4-50.2
"IX_HCD_SST_CLA_POI_2_SEL"	I 1078.5	BOOL	// Spannhydraulik Anwahl Spannkreis 2   /H4-50.5
"IX_CC_RAKE_1_REAR"	I 1080.0	BOOL	// Spaenefoerderer -Rechen 1 Hubeinheit hinten
"IX_CC_RAKE_1_FRONT"	I 1080.1	BOOL	// Spaenefoerderer -Rechen 1 Hubeinheit vorn
"IX_CC_RAKE_2_REAR"	I 1080.2	BOOL	// Spaenefoerderer -Rechen 2 Hubeinheit hinten
"IX_CC_RAKE_2_FRONT"	I 1080.3	BOOL	// Spaenefoerderer -Rechen 2 Hubeinheit vorn
"IX_CC_RAKE_UNPRESS"	I 1080.4	BOOL	// Druckschalter Hauptluft Spaenefoerderer-Rechen
"IX_CC_RAKE_UNPRESS_D"	I 1080.5	BOOL	// Diagnose Druckschalter Hauptluft Spaenefoerderer-Rechen
"IX_HCD_MPL_ENGAGED"	I 1085.0	BOOL	// Hydraulik Maschinenplatz Kupplung angekuppelt   /H4-07.3
"IX_HCD_MPL_DISENGAGED"	I 1085.1	BOOL	// Hydraulik Maschinenplatz Kupplung abgekuppelt   /H4-07.3
"IX_WW_GRF_ENTRIEGELT"	I 1117.3	BOOL	// Verriegelung Werkzeuggreifer entriegelt
"IX_PC_MPL_MCON_DENGD"	I 1117.4	BOOL	// Medienkupplung Fraes-Drehtisch eingefahren
"IX_PC_MPL_MCON_ENGAGED"	I 1117.5	BOOL	// Medienkupplung Fraes-Drehtisch ausgefahren
"IX_CC_NIVEAU_MAX_N"	I 1117.6	BOOL	// Spaenefoerderer Ueberlaufbegrenzung Sammelbehaelter
"IX_FMS_APC_MOVEMENT_OK"	I 1150.1	BOOL	// Handlingsystem MC INPUT Byte 1 Bit 1 Handlingsystem APC movement ok
"IX_FMS_CNC_START"	I 1150.2	BOOL	// Handlingsystem MC INPUT Byte 1 Bit 2 CNC Start
"IX_FMS_AUTO_POWER_OFF"	I 1150.3	BOOL	// Handlingsystem MC INPUT Byte 1 Bit 3 Auto Power  Off
"IX_FMS_FIXTURE_RELEASE"	I 1150.4	BOOL	// Handlingsystem MC INPUT Byte 1 Bit 4
"IX_GEN_OM_ID_SYNC"	I 1151.0	BOOL	// Smartkey: Zeigt den START und RESTART der übertragung an (>50ms)
"IX_GEN_OM_ID_CLOCK"	I 1151.1	BOOL	// Smartkey: Protokoll-Taktrate. Daten können gelesen werden
"IX_GEN_OM_ID_DATA_0"	I 1151.2	BOOL	// Smartkey: Daten – Spur 1
"IX_GEN_OM_ID_DATA_1"	I 1151.3	BOOL	// Smartkey: Daten – Spur 2
"IX_SST_SPEED_RPM_BIT_1"	I 1200.0	BOOL
"IX_SST_SPEED_RPM_BIT_2"	I 1200.1	BOOL
"IX_SST_SPEED_RPM_BIT_3"	I 1200.2	BOOL
"IX_SST_SPEED_RPM_BIT_4"	I 1200.3	BOOL
"IX_SPI_TEMP_RDY"	I 2010.0	BOOL	// Temperaturüberwachung Motorspindel (55/65H)
"IX_PC_MPL_PALLET_CLPED_D"	I 2010.1	BOOL	// Diagnose Palettenklemmung geklemmt  (55/65H)
"IX_PC_MPL_PALLET_RELD_D"	I 2010.2	BOOL	// Diagnose Palettenklemmung geloest (55/65H)
"IX_PC_MPL_OCCUPIED_D"	I 2010.3	BOOL	// Diagnose Palette Maschine vorhanden (55/65H)
"IX_GEN_HYD_PRESSURE_OK_D"	I 2010.4	BOOL	// Diagnose Druckueberwachung Hydraulik (55/65H)
"IX_GEN_CAIR_PRE_OK_D"	I 2010.5	BOOL	// Diagnose Druckueberwachung Pneumatik (55/65H)
"IX_CU_GAP_SCREEN_CL_UPP"	I 2010.7	BOOL	// Kühlmittelanlage Spaltsieb oben
"IX_CU_GAP_SCREEN_CL_LOW"	I 2011.0	BOOL	// Kühlmittelanlage Spaltsieb unten
"IX_CU_NEG_PRESS_MONITOR"	I 2011.1	BOOL	// Kühlmittelanlage Spaltsieb unten
"IX_TM_PUMP_MPS"	I 2011.2	BOOL	// Motorschutzschalter Hebepumpe Werkzeugmagazin
"IX_TM_PUMP_ON"	I 2011.3	BOOL	// Hebepumpe Werkzeugmagazin ein
"IX_CU_FLUSH_PIST_SST_ON"	I 2011.4	BOOL	// Spuelpistole Ruestplatz ein
"IX_TC_POSITION_BRUSH_CLE"	I 2011.5	BOOL	// Positionsueberwachung Reinigung Werkzeugkegel
"IX_TORQ_PROP_FILL_MON"	I 2011.6	BOOL	// Fuellstand Oelbehaelter Drehmomentstuetze
"IX_CU_M7_PRESSURE0_ON"	I 2030.1	BOOL
"IX_CU_M7_PRESSURE2_ON"	I 2030.2	BOOL
"IX_SST_BUTTON_FLUSH_ON"	I 3040.6	BOOL	// B2-87.4 Taste Aktivierung Spuelung Ruestplatz
"IX_SST_SUPP_CHECK_OFF"	I 3040.7	BOOL	// Schlüsselschalter Auflagekontrolle aus
"IX_SST_DOOR_1_OPENED"	I 3041.6	BOOL	// G1-94.5 Rüstplatz-Tür 1 ist offen
"IX_SST_DOOR_2_OPENED"	I 3041.7	BOOL	// G1-94.5 Rüstplatz-Tür 2 ist offen
"IX_GEN_POWERFAIL_MONITOR"	I 3047.0	BOOL	// A0-82.4 Spannungsüberwachung Netz nicht in Ordnung
"IX_ROBOT_LOCK"	I 3048.1	BOOL	// F4-66.2 Schlüsselschalter Betriebsart Roboter gesperrt
"IX_SST_SC_CL_PO_1_ACT"	I 3073.0	BOOL	// H4-95.2 Auflagenkontrolle Spannstelle 1 gespannt OK
"IX_SST_SC_CL_PO_2_ACT"	I 3073.1	BOOL	// H4-95.5 Auflagenkontrolle Spannstelle 2 gespannt OK
